LIN {X 0,Y 657.537,Z 599.865,A -85,B 0,C 180,E1 28395.268,E2 28395.268} C_VEL
LIN {X 0,Y 653.321,Z 821.185,A -85,B 0,C 180,E1 28392.316,E2 28392.316} C_VEL
LIN {X 0,Y 652.432,Z 844.585,A -85,B 0,C 180,E1 28391.93,E2 28391.93} C_VEL
LIN {X 0,Y 651.296,Z 867.25,A -85,B 0,C 180,E1 28391.436,E2 28391.436} C_VEL
LIN {X 0,Y 649.719,Z 893.344,A -85,B 0,C 180,E1 28390.715,E2 28390.715} C_VEL
LIN {X 0,Y 647.795,Z 918.743,A -85,B 0,C 180,E1 28389.832,E2 28389.832} C_VEL
LIN {X 0,Y 645.973,Z 940.605,A -85,B 0,C 180,E1 28388.933,E2 28388.933} C_VEL
LIN {X 0,Y 644.086,Z 961.718,A -85,B 0,C 180,E1 28387.933,E2 28387.933} C_VEL
LIN {X 0,Y 641.744,Z 986.523,A -85,B 0,C 180,E1 28386.58,E2 28386.58} C_VEL
LIN {X 0,Y 639.474,Z 1008.599,A -85,B 0,C 180,E1 28385.182,E2 28385.182} C_VEL
LIN {X 0,Y 637.565,Z 1026.909,A -85,B 0,C 180,E1 28383.884,E2 28383.884} C_VEL
LIN {X 0,Y 635.698,Z 1044.667,A -85,B 0,C 180,E1 28382.488,E2 28382.488} C_VEL
LIN {X 0,Y 633.545,Z 1065.498,A -85,B 0,C 180,E1 28380.667,E2 28380.667} C_VEL
LIN {X 0,Y 631.511,Z 1085.195,A -85,B 0,C 180,E1 28378.697,E2 28378.697} C_VEL
LIN {X 0,Y 630.035,Z 1100.537,A -85,B 0,C 180,E1 28376.993,E2 28376.993} C_VEL
LIN {X 0,Y 628.438,Z 1118.013,A -85,B 0,C 180,E1 28374.836,E2 28374.836} C_VEL
LIN {X 0,Y 627.118,Z 1133.831,A -85,B 0,C 180,E1 28372.597,E2 28372.597} C_VEL
LIN {X 0,Y 626.191,Z 1146.584,A -85,B 0,C 180,E1 28370.566,E2 28370.566} C_VEL
LIN {X 0,Y 625.357,Z 1159.892,A -85,B 0,C 180,E1 28368.166,E2 28368.166} C_VEL
LIN {X 0,Y 624.743,Z 1171.081,A -85,B 0,C 180,E1 28365.788,E2 28365.788} C_VEL
LIN {X 0,Y 624.416,Z 1179.161,A -85,B 0,C 180,E1 28363.803,E2 28363.803} C_VEL
LIN {X 0,Y 624.174,Z 1186.707,A -85,B 0,C 180,E1 28361.644,E2 28361.644} C_VEL
LIN {X 0,Y 624.016,Z 1193.595,A -85,B 0,C 180,E1 28359.22,E2 28359.22} C_VEL
LIN {X 0,Y 623.938,Z 1198.919,A -85,B 0,C 180,E1 28356.718,E2 28356.718} C_VEL
LIN {X 0,Y 623.914,Z 1202.24,A -85,B 0,C 180,E1 28354.504,E2 28354.504} C_VEL
LIN {X 0,Y 623.912,Z 1204.382,A -85,B 0,C 180,E1 28352.112,E2 28352.112} C_VEL
LIN {X 0,Y 623.892,Z 1204.894,A -85,B 0,C 180,E1 28349.541,E2 28349.541} C_VEL
LIN {X 0,Y 623.91,Z 1204.004,A -85,B 0,C 180,E1 28347.336,E2 28347.336} C_VEL
LIN {X 0,Y 623.923,Z 1201.671,A -85,B 0,C 180,E1 28345.036,E2 28345.036} C_VEL
LIN {X 0,Y 623.958,Z 1197.542,A -85,B 0,C 180,E1 28342.542,E2 28342.542} C_VEL
LIN {X 0,Y 624.046,Z 1191.872,A -85,B 0,C 180,E1 28340.129,E2 28340.129} C_VEL
LIN {X 0,Y 624.21,Z 1184.888,A -85,B 0,C 180,E1 28337.793,E2 28337.793} C_VEL
LIN {X 0,Y 624.578,Z 1175.442,A -85,B 0,C 180,E1 28335.229,E2 28335.229} C_VEL
LIN {X 0,Y 625.049,Z 1164.999,A -85,B 0,C 180,E1 28332.882,E2 28332.882} C_VEL
LIN {X 0,Y 625.664,Z 1154.466,A -85,B 0,C 180,E1 28330.821,E2 28330.821} C_VEL
LIN {X 0,Y 626.613,Z 1140.788,A -85,B 0,C 180,E1 28328.469,E2 28328.469} C_VEL
LIN {X 0,Y 627.822,Z 1125.096,A -85,B 0,C 180,E1 28326.139,E2 28326.139} C_VEL
LIN {X 0,Y 629.061,Z 1111.084,A -85,B 0,C 180,E1 28324.284,E2 28324.284} C_VEL
LIN {X 0,Y 630.771,Z 1092.863,A -85,B 0,C 180,E1 28322.12,E2 28322.12} C_VEL
LIN {X 0,Y 632.663,Z 1073.815,A -85,B 0,C 180,E1 28320.144,E2 28320.144} C_VEL
LIN {X 0,Y 634.36,Z 1057.393,A -85,B 0,C 180,E1 28318.606,E2 28318.606} C_VEL
LIN {X 0,Y 636.318,Z 1038.641,A -85,B 0,C 180,E1 28317.018,E2 28317.018} C_VEL
LIN {X 0,Y 638.857,Z 1014.539,A -85,B 0,C 180,E1 28315.223,E2 28315.223} C_VEL
LIN {X 0,Y 640.898,Z 994.594,A -85,B 0,C 180,E1 28313.916,E2 28313.916} C_VEL
LIN {X 0,Y 642.854,Z 974.951,A -85,B 0,C 180,E1 28312.769,E2 28312.769} C_VEL
LIN {X 0,Y 645.083,Z 951.673,A -85,B 0,C 180,E1 28311.572,E2 28311.572} C_VEL
LIN {X 0,Y 647.292,Z 925.381,A -85,B 0,C 180,E1 28310.428,E2 28310.428} C_VEL
LIN {X 0,Y 648.897,Z 904.132,A -85,B 0,C 180,E1 28309.643,E2 28309.643} C_VEL
LIN {X 0,Y 650.369,Z 882.585,A -85,B 0,C 180,E1 28308.97,E2 28308.97} C_VEL
LIN {X 0,Y 651.781,Z 858.661,A -85,B 0,C 180,E1 28308.36,E2 28308.36} C_VEL
LIN {X 0,Y 653.042,Z 830.092,A -85,B 0,C 180,E1 28307.816,E2 28307.816} C_VEL
LIN {X 0,Y 654.465,Z 762.422,A -85,B 0,C 180,E1 28306.902,E2 28306.902} C_VEL
LIN {X 0,Y 658.724,Z 539.813,A -85,B 0,C 180,E1 28303.919,E2 28303.919} C_VEL
LIN {X 0,Y 661.621,Z 393.143,A -85,B 0,C 180,E1 28301.897,E2 28301.897} C_VEL
LIN {X 0,Y 647.792,Z 372.953,A -85,B 0,C 180,E1 28300.181,E2 28300.181} C_VEL
LIN {X 0,Y 638.276,Z 359.45,A -85,B 0,C 180,E1 28298.917,E2 28298.917} C_VEL
LIN {X 0,Y 631.39,Z 349.683,A -85,B 0,C 180,E1 28297.912,E2 28297.912} C_VEL
LIN {X 0,Y 627.324,Z 341.452,A -85,B 0,C 180,E1 28296.593,E2 28296.593} C_VEL
LIN {X 0,Y 625.216,Z 337.776,A -85,B 0,C 180,E1 28295.94,E2 28295.94} C_VEL
LIN {X 0,Y 624.896,Z 336.388,A -85,B 0,C 180,E1 28295.735,E2 28295.735} C_VEL
LIN {X 0,Y 624.89,Z 336.391,A -85,B 0,C 180,E1 28292.959,E2 28292.959} C_VEL
LIN {X 0,Y 624.914,Z 336.381,A -85,B 0,C 180,E1 28289.737,E2 28289.737} C_VEL
LIN {X 0,Y 624.88,Z 336.358,A -85,B 0,C 180,E1 28286.97,E2 28286.97} C_VEL
LIN {X 0,Y 624.953,Z 336.372,A -85,B 0,C 180,E1 28283.878,E2 28283.878} C_VEL
LIN {X 0,Y 624.884,Z 336.384,A -85,B 0,C 180,E1 28280.906,E2 28280.906} C_VEL
LIN {X 0,Y 624.944,Z 336.356,A -85,B 0,C 180,E1 28277.987,E2 28277.987} C_VEL
LIN {X 0,Y 624.888,Z 336.391,A -85,B 0,C 180,E1 28274.887,E2 28274.887} C_VEL
LIN {X 0,Y 624.922,Z 336.352,A -85,B 0,C 180,E1 28272.005,E2 28272.005} C_VEL
LIN {X 0,Y 624.895,Z 336.385,A -85,B 0,C 180,E1 28268.836,E2 28268.836} C_VEL
LIN {X 0,Y 624.901,Z 336.36,A -85,B 0,C 180,E1 28266.062,E2 28266.062} C_VEL
LIN {X 0,Y 624.901,Z 336.375,A -85,B 0,C 180,E1 28262.751,E2 28262.751} C_VEL
LIN {X 0,Y 624.902,Z 336.375,A -85,B 0,C 180,E1 28259.908,E2 28259.908} C_VEL
LIN {X 0,Y 624.903,Z 336.36,A -85,B 0,C 180,E1 28256.606,E2 28256.606} C_VEL
LIN {X 0,Y 624.903,Z 336.384,A -85,B 0,C 180,E1 28253.754,E2 28253.754} C_VEL
LIN {X 0,Y 624.912,Z 336.355,A -85,B 0,C 180,E1 28250.514,E2 28250.514} C_VEL
LIN {X 0,Y 624.902,Z 336.388,A -85,B 0,C 180,E1 28247.619,E2 28247.619} C_VEL
LIN {X 0,Y 624.921,Z 336.363,A -85,B 0,C 180,E1 28244.404,E2 28244.404} C_VEL
LIN {X 0,Y 624.897,Z 336.37,A -85,B 0,C 180,E1 28241.529,E2 28241.529} C_VEL
LIN {X 0,Y 624.942,Z 336.389,A -85,B 0,C 180,E1 28238.365,E2 28238.365} C_VEL
LIN {X 0,Y 624.894,Z 336.369,A -85,B 0,C 180,E1 28235.416,E2 28235.416} C_VEL
LIN {X 0,Y 624.956,Z 336.386,A -85,B 0,C 180,E1 28232.355,E2 28232.355} C_VEL
LIN {X 0,Y 624.976,Z 336.514,A -85,B 0,C 180,E1 28230.372,E2 28230.372} C_VEL
LIN {X 0,Y 626.376,Z 340.092,A -85,B 0,C 180,E1 28229.812,E2 28229.812} C_VEL
LIN {X 0,Y 627.464,Z 341.921,A -85,B 0,C 180,E1 28229.499,E2 28229.499} C_VEL
LIN {X 0,Y 630.591,Z 346.07,A -85,B 0,C 180,E1 28229.033,E2 28229.033} C_VEL
LIN {X 0,Y 642.353,Z 362.019,A -85,B 0,C 180,E1 28227.386,E2 28227.386} C_VEL
LIN {X 0,Y 655.331,Z 380.655,A -85,B 0,C 180,E1 28225.722,E2 28225.722} C_VEL
LIN {X 0,Y 661.575,Z 390.24,A -85,B 0,C 180,E1 28224.954,E2 28224.954} C_VEL
LIN {X 0,Y 659.29,Z 501.464,A -85,B 0,C 180,E1 28223.422,E2 28223.422} C_VEL
LIN {X 0,Y 658.447,Z 509.169,A -85,B 0,C 180,E1 28223.38,E2 28223.38} C_VEL
LIN {X 0,Y 653.685,Z 529.837,A -85,B 0,C 180,E1 28223.497,E2 28223.497} C_VEL
LIN {X 0,Y 653.027,Z 536.446,A -85,B 0,C 180,E1 28223.454,E2 28223.454} C_VEL
LIN {X 0,Y 648.61,Z 753.058,A -85,B 0,C 180,E1 28220.529,E2 28220.529} C_VEL
LIN {X 0,Y 647.089,Z 821.836,A -85,B 0,C 180,E1 28219.592,E2 28219.592} C_VEL
LIN {X 0,Y 645.779,Z 848.344,A -85,B 0,C 180,E1 28219.075,E2 28219.075} C_VEL
LIN {X 0,Y 644.398,Z 870.837,A -85,B 0,C 180,E1 28218.507,E2 28218.507} C_VEL
LIN {X 0,Y 642.785,Z 893.737,A -85,B 0,C 180,E1 28217.797,E2 28217.797} C_VEL
LIN {X 0,Y 640.614,Z 920.334,A -85,B 0,C 180,E1 28216.793,E2 28216.793} C_VEL
LIN {X 0,Y 638.585,Z 942.122,A -85,B 0,C 180,E1 28215.816,E2 28215.816} C_VEL
LIN {X 0,Y 636.483,Z 963.279,A -85,B 0,C 180,E1 28214.73,E2 28214.73} C_VEL
LIN {X 0,Y 633.956,Z 987.267,A -85,B 0,C 180,E1 28213.32,E2 28213.32} C_VEL
LIN {X 0,Y 631.38,Z 1010.175,A -85,B 0,C 180,E1 28211.763,E2 28211.763} C_VEL
LIN {X 0,Y 628.962,Z 1032.056,A -85,B 0,C 180,E1 28210.078,E2 28210.078} C_VEL
LIN {X 0,Y 626.551,Z 1053.456,A -85,B 0,C 180,E1 28208.198,E2 28208.198} C_VEL
LIN {X 0,Y 624.312,Z 1073.834,A -85,B 0,C 180,E1 28206.176,E2 28206.176} C_VEL
LIN {X 0,Y 622.264,Z 1093.517,A -85,B 0,C 180,E1 28203.948,E2 28203.948} C_VEL
LIN {X 0,Y 620.561,Z 1111.006,A -85,B 0,C 180,E1 28201.706,E2 28201.706} C_VEL
LIN {X 0,Y 619.125,Z 1127.45,A -85,B 0,C 180,E1 28199.295,E2 28199.295} C_VEL
LIN {X 0,Y 618.008,Z 1142.104,A -85,B 0,C 180,E1 28196.833,E2 28196.833} C_VEL
LIN {X 0,Y 617.161,Z 1155.043,A -85,B 0,C 180,E1 28194.299,E2 28194.299} C_VEL
LIN {X 0,Y 616.625,Z 1165.506,A -85,B 0,C 180,E1 28191.897,E2 28191.897} C_VEL
LIN {X 0,Y 616.242,Z 1174.897,A -85,B 0,C 180,E1 28189.329,E2 28189.329} C_VEL
LIN {X 0,Y 616.066,Z 1181.779,A -85,B 0,C 180,E1 28186.986,E2 28186.986} C_VEL
LIN {X 0,Y 615.973,Z 1187.229,A -85,B 0,C 180,E1 28184.653,E2 28184.653} C_VEL
LIN {X 0,Y 615.925,Z 1191.546,A -85,B 0,C 180,E1 28182.088,E2 28182.088} C_VEL
LIN {X 0,Y 615.913,Z 1193.955,A -85,B 0,C 180,E1 28179.72,E2 28179.72} C_VEL
LIN {X 0,Y 615.896,Z 1194.864,A -85,B 0,C 180,E1 28177.556,E2 28177.556} C_VEL
LIN {X 0,Y 615.914,Z 1194.562,A -85,B 0,C 180,E1 28175.123,E2 28175.123} C_VEL
LIN {X 0,Y 615.916,Z 1192.49,A -85,B 0,C 180,E1 28172.605,E2 28172.605} C_VEL
LIN {X 0,Y 615.946,Z 1189.149,A -85,B 0,C 180,E1 28170.279,E2 28170.279} C_VEL
LIN {X 0,Y 616.031,Z 1183.731,A -85,B 0,C 180,E1 28167.675,E2 28167.675} C_VEL
LIN {X 0,Y 616.189,Z 1176.982,A -85,B 0,C 180,E1 28165.253,E2 28165.253} C_VEL
LIN {X 0,Y 616.445,Z 1169.355,A -85,B 0,C 180,E1 28163.013,E2 28163.013} C_VEL
LIN {X 0,Y 616.94,Z 1159.075,A -85,B 0,C 180,E1 28160.485,E2 28160.485} C_VEL
LIN {X 0,Y 617.683,Z 1146.755,A -85,B 0,C 180,E1 28157.947,E2 28157.947} C_VEL
LIN {X 0,Y 618.726,Z 1132.355,A -85,B 0,C 180,E1 28155.399,E2 28155.399} C_VEL
LIN {X 0,Y 620.085,Z 1116.227,A -85,B 0,C 180,E1 28152.934,E2 28152.934} C_VEL
LIN {X 0,Y 621.745,Z 1098.393,A -85,B 0,C 180,E1 28150.556,E2 28150.556} C_VEL
LIN {X 0,Y 623.702,Z 1079.651,A -85,B 0,C 180,E1 28148.364,E2 28148.364} C_VEL
LIN {X 0,Y 625.944,Z 1058.763,A -85,B 0,C 180,E1 28146.213,E2 28146.213} C_VEL
LIN {X 0,Y 628.328,Z 1037.643,A -85,B 0,C 180,E1 28144.302,E2 28144.302} C_VEL
LIN {X 0,Y 630.948,Z 1014.168,A -85,B 0,C 180,E1 28142.437,E2 28142.437} C_VEL
LIN {X 0,Y 633.461,Z 991.448,A -85,B 0,C 180,E1 28140.861,E2 28140.861} C_VEL
LIN {X 0,Y 636.2,Z 966.176,A -85,B 0,C 180,E1 28139.337,E2 28139.337} C_VEL
LIN {X 0,Y 638.384,Z 944.2,A -85,B 0,C 180,E1 28138.195,E2 28138.195} C_VEL
LIN {X 0,Y 640.435,Z 922.22,A -85,B 0,C 180,E1 28137.198,E2 28137.198} C_VEL
LIN {X 0,Y 642.615,Z 896.084,A -85,B 0,C 180,E1 28136.191,E2 28136.191} C_VEL
LIN {X 0,Y 644.347,Z 871.789,A -85,B 0,C 180,E1 28135.431,E2 28135.431} C_VEL
LIN {X 0,Y 645.709,Z 849.449,A -85,B 0,C 180,E1 28134.86,E2 28134.86} C_VEL
LIN {X 0,Y 646.986,Z 824.075,A -85,B 0,C 180,E1 28134.355,E2 28134.355} C_VEL
LIN {X 0,Y 648.108,Z 779.029,A -85,B 0,C 180,E1 28133.727,E2 28133.727} C_VEL
LIN {X 0,Y 652.675,Z 553.676,A -85,B 0,C 180,E1 28130.693,E2 28130.693} C_VEL
LIN {X 0,Y 656.073,Z 393.886,A -85,B 0,C 180,E1 28128.478,E2 28128.478} C_VEL
LIN {X 0,Y 644.814,Z 377.11,A -85,B 0,C 180,E1 28127.047,E2 28127.047} C_VEL
LIN {X 0,Y 633.812,Z 361.802,A -85,B 0,C 180,E1 28125.582,E2 28125.582} C_VEL
LIN {X 0,Y 626.174,Z 351.738,A -85,B 0,C 180,E1 28124.54,E2 28124.54} C_VEL
LIN {X 0,Y 622.262,Z 346.503,A -85,B 0,C 180,E1 28123.993,E2 28123.993} C_VEL
LIN {X 0,Y 618.866,Z 341.624,A -85,B 0,C 180,E1 28123.494,E2 28123.494} C_VEL
LIN {X 0,Y 617.209,Z 338.714,A -85,B 0,C 180,E1 28123.003,E2 28123.003} C_VEL
LIN {X 0,Y 616.913,Z 337.36,A -85,B 0,C 180,E1 28122.807,E2 28122.807} C_VEL
LIN {X 0,Y 616.952,Z 337.385,A -85,B 0,C 180,E1 28120.047,E2 28120.047} C_VEL
LIN {X 0,Y 616.924,Z 337.379,A -85,B 0,C 180,E1 28116.848,E2 28116.848} C_VEL
LIN {X 0,Y 616.932,Z 337.375,A -85,B 0,C 180,E1 28114.089,E2 28114.089} C_VEL
LIN {X 0,Y 616.933,Z 337.382,A -85,B 0,C 180,E1 28110.8,E2 28110.8} C_VEL
LIN {X 0,Y 616.92,Z 337.342,A -85,B 0,C 180,E1 28108.141,E2 28108.141} C_VEL
LIN {X 0,Y 616.979,Z 337.38,A -85,B 0,C 180,E1 28105.023,E2 28105.023} C_VEL
LIN {X 0,Y 616.916,Z 337.342,A -85,B 0,C 180,E1 28102.188,E2 28102.188} C_VEL
LIN {X 0,Y 616.993,Z 337.368,A -85,B 0,C 180,E1 28099.207,E2 28099.207} C_VEL
LIN {X 0,Y 616.923,Z 337.376,A -85,B 0,C 180,E1 28096.187,E2 28096.187} C_VEL
LIN {X 0,Y 616.941,Z 337.373,A -85,B 0,C 180,E1 28093.493,E2 28093.493} C_VEL
LIN {X 0,Y 616.939,Z 337.369,A -85,B 0,C 180,E1 28090.27,E2 28090.27} C_VEL
LIN {X 0,Y 616.931,Z 337.381,A -85,B 0,C 180,E1 28087.544,E2 28087.544} C_VEL
LIN {X 0,Y 616.981,Z 337.377,A -85,B 0,C 180,E1 28084.462,E2 28084.462} C_VEL
LIN {X 0,Y 616.924,Z 337.377,A -85,B 0,C 180,E1 28081.579,E2 28081.579} C_VEL
LIN {X 0,Y 617.008,Z 337.365,A -85,B 0,C 180,E1 28078.607,E2 28078.607} C_VEL
LIN {X 0,Y 616.926,Z 337.368,A -85,B 0,C 180,E1 28075.538,E2 28075.538} C_VEL
LIN {X 0,Y 616.981,Z 337.371,A -85,B 0,C 180,E1 28072.644,E2 28072.644} C_VEL
LIN {X 0,Y 616.934,Z 337.376,A -85,B 0,C 180,E1 28069.541,E2 28069.541} C_VEL
LIN {X 0,Y 616.953,Z 337.333,A -85,B 0,C 180,E1 28066.695,E2 28066.695} C_VEL
LIN {X 0,Y 616.945,Z 337.378,A -85,B 0,C 180,E1 28063.523,E2 28063.523} C_VEL
LIN {X 0,Y 616.934,Z 337.337,A -85,B 0,C 180,E1 28060.791,E2 28060.791} C_VEL
LIN {X 0,Y 616.97,Z 337.375,A -85,B 0,C 180,E1 28057.613,E2 28057.613} C_VEL
LIN {X 0,Y 616.931,Z 337.34,A -85,B 0,C 180,E1 28054.77,E2 28054.77} C_VEL
LIN {X 0,Y 616.996,Z 337.367,A -85,B 0,C 180,E1 28051.635,E2 28051.635} C_VEL
LIN {X 0,Y 616.934,Z 337.374,A -85,B 0,C 180,E1 28048.759,E2 28048.759} C_VEL
LIN {X 0,Y 617.011,Z 337.376,A -85,B 0,C 180,E1 28045.735,E2 28045.735} C_VEL
LIN {X 0,Y 616.961,Z 337.53,A -85,B 0,C 180,E1 28044.876,E2 28044.876} C_VEL
LIN {X 0,Y 618.247,Z 340.864,A -85,B 0,C 180,E1 28044.392,E2 28044.392} C_VEL
LIN {X 0,Y 619.292,Z 342.381,A -85,B 0,C 180,E1 28044.12,E2 28044.12} C_VEL
LIN {X 0,Y 623.249,Z 350.426,A -85,B 0,C 180,E1 28042.927,E2 28042.927} C_VEL
LIN {X 0,Y 633.099,Z 363.839,A -85,B 0,C 180,E1 28041.57,E2 28041.57} C_VEL
LIN {X 0,Y 642.371,Z 376.815,A -85,B 0,C 180,E1 28040.328,E2 28040.328} C_VEL
LIN {X 0,Y 654.585,Z 394.719,A -85,B 0,C 180,E1 28038.767,E2 28038.767} C_VEL
LIN {X 0,Y 656.243,Z 397.52,A -85,B 0,C 180,E1 28038.557,E2 28038.557} C_VEL
LIN {X 0,Y 651.839,Z 602.931,A -85,B 0,C 180,E1 28035.728,E2 28035.728} C_VEL
LIN {X 0,Y 647.36,Z 822.437,A -85,B 0,C 180,E1 28032.775,E2 28032.775} C_VEL
LIN {X 0,Y 646.442,Z 845.047,A -85,B 0,C 180,E1 28032.397,E2 28032.397} C_VEL
LIN {X 0,Y 645.242,Z 867.553,A -85,B 0,C 180,E1 28031.903,E2 28031.903} C_VEL
LIN {X 0,Y 643.563,Z 893.754,A -85,B 0,C 180,E1 28031.174,E2 28031.174} C_VEL
LIN {X 0,Y 641.555,Z 918.74,A -85,B 0,C 180,E1 28030.299,E2 28030.299} C_VEL
LIN {X 0,Y 639.694,Z 939.866,A -85,B 0,C 180,E1 28029.427,E2 28029.427} C_VEL
LIN {X 0,Y 637.715,Z 960.71,A -85,B 0,C 180,E1 28028.437,E2 28028.437} C_VEL
LIN {X 0,Y 635.358,Z 983.923,A -85,B 0,C 180,E1 28027.178,E2 28027.178} C_VEL
LIN {X 0,Y 632.763,Z 1007.862,A -85,B 0,C 180,E1 28025.667,E2 28025.667} C_VEL
LIN {X 0,Y 630.635,Z 1026.957,A -85,B 0,C 180,E1 28024.303,E2 28024.303} C_VEL
LIN {X 0,Y 628.619,Z 1044.936,A -85,B 0,C 180,E1 28022.876,E2 28022.876} C_VEL
LIN {X 0,Y 626.328,Z 1065.691,A -85,B 0,C 180,E1 28021.04,E2 28021.04} C_VEL
LIN {X 0,Y 624.159,Z 1084.994,A -85,B 0,C 180,E1 28019.09,E2 28019.09} C_VEL
LIN {X 0,Y 622.55,Z 1100.535,A -85,B 0,C 180,E1 28017.344,E2 28017.344} C_VEL
LIN {X 0,Y 620.832,Z 1118.042,A -85,B 0,C 180,E1 28015.158,E2 28015.158} C_VEL
LIN {X 0,Y 619.41,Z 1133.833,A -85,B 0,C 180,E1 28012.894,E2 28012.894} C_VEL
LIN {X 0,Y 618.402,Z 1146.582,A -85,B 0,C 180,E1 28010.837,E2 28010.837} C_VEL
LIN {X 0,Y 617.488,Z 1159.949,A -85,B 0,C 180,E1 28008.394,E2 28008.394} C_VEL
LIN {X 0,Y 616.833,Z 1171.082,A -85,B 0,C 180,E1 28005.995,E2 28005.995} C_VEL
LIN {X 0,Y 616.461,Z 1179.162,A -85,B 0,C 180,E1 28003.985,E2 28003.985} C_VEL
LIN {X 0,Y 616.199,Z 1186.401,A -85,B 0,C 180,E1 28001.892,E2 28001.892} C_VEL
LIN {X 0,Y 616.035,Z 1193.353,A -85,B 0,C 180,E1 27999.435,E2 27999.435} C_VEL
LIN {X 0,Y 615.943,Z 1198.756,A -85,B 0,C 180,E1 27996.899,E2 27996.899} C_VEL
LIN {X 0,Y 615.914,Z 1202.2,A -85,B 0,C 180,E1 27994.593,E2 27994.593} C_VEL
LIN {X 0,Y 615.911,Z 1204.326,A -85,B 0,C 180,E1 27992.233,E2 27992.233} C_VEL
LIN {X 0,Y 615.894,Z 1204.917,A -85,B 0,C 180,E1 27989.628,E2 27989.628} C_VEL
LIN {X 0,Y 615.911,Z 1204.001,A -85,B 0,C 180,E1 27987.302,E2 27987.302} C_VEL
LIN {X 0,Y 615.925,Z 1201.668,A -85,B 0,C 180,E1 27984.971,E2 27984.971} C_VEL
LIN {X 0,Y 615.96,Z 1197.542,A -85,B 0,C 180,E1 27982.445,E2 27982.445} C_VEL
LIN {X 0,Y 616.061,Z 1191.869,A -85,B 0,C 180,E1 27979.999,E2 27979.999} C_VEL
LIN {X 0,Y 616.231,Z 1185.188,A -85,B 0,C 180,E1 27977.728,E2 27977.728} C_VEL
LIN {X 0,Y 616.603,Z 1176.301,A -85,B 0,C 180,E1 27975.251,E2 27975.251} C_VEL
LIN {X 0,Y 617.134,Z 1165.456,A -85,B 0,C 180,E1 27972.753,E2 27972.753} C_VEL
LIN {X 0,Y 617.794,Z 1154.968,A -85,B 0,C 180,E1 27970.662,E2 27970.662} C_VEL
LIN {X 0,Y 618.708,Z 1142.537,A -85,B 0,C 180,E1 27968.479,E2 27968.479} C_VEL
LIN {X 0,Y 620.047,Z 1126.495,A -85,B 0,C 180,E1 27966.023,E2 27966.023} C_VEL
LIN {X 0,Y 621.426,Z 1111.852,A -85,B 0,C 180,E1 27964.047,E2 27964.047} C_VEL
LIN {X 0,Y 623.059,Z 1095.44,A -85,B 0,C 180,E1 27962.057,E2 27962.057} C_VEL
LIN {X 0,Y 625.236,Z 1075.26,A -85,B 0,C 180,E1 27959.904,E2 27959.904} C_VEL
LIN {X 0,Y 627.085,Z 1058.502,A -85,B 0,C 180,E1 27958.307,E2 27958.307} C_VEL
LIN {X 0,Y 629.038,Z 1041.012,A -85,B 0,C 180,E1 27956.799,E2 27956.799} C_VEL
LIN {X 0,Y 631.555,Z 1018.937,A -85,B 0,C 180,E1 27955.096,E2 27955.096} C_VEL
LIN {X 0,Y 634.035,Z 996.25,A -85,B 0,C 180,E1 27953.578,E2 27953.578} C_VEL
LIN {X 0,Y 636.01,Z 977.648,A -85,B 0,C 180,E1 27952.47,E2 27952.47} C_VEL
LIN {X 0,Y 638.028,Z 957.699,A -85,B 0,C 180,E1 27951.413,E2 27951.413} C_VEL
LIN {X 0,Y 640.077,Z 936.082,A -85,B 0,C 180,E1 27950.407,E2 27950.407} C_VEL
LIN {X 0,Y 642.391,Z 908.567,A -85,B 0,C 180,E1 27949.325,E2 27949.325} C_VEL
LIN {X 0,Y 644.095,Z 885.248,A -85,B 0,C 180,E1 27948.574,E2 27948.574} C_VEL
LIN {X 0,Y 645.474,Z 863.386,A -85,B 0,C 180,E1 27947.996,E2 27947.996} C_VEL
LIN {X 0,Y 646.71,Z 839.526,A -85,B 0,C 180,E1 27947.497,E2 27947.497} C_VEL
LIN {X 0,Y 647.823,Z 804.077,A -85,B 0,C 180,E1 27946.972,E2 27946.972} C_VEL
LIN {X 0,Y 652.338,Z 579.129,A -85,B 0,C 180,E1 27943.949,E2 27943.949} C_VEL
LIN {X 0,Y 656.196,Z 397.117,A -85,B 0,C 180,E1 27941.433,E2 27941.433} C_VEL
LIN {X 0,Y 643.844,Z 378.961,A -85,B 0,C 180,E1 27939.867,E2 27939.867} C_VEL
LIN {X 0,Y 634.511,Z 365.563,A -85,B 0,C 180,E1 27938.594,E2 27938.594} C_VEL
LIN {X 0,Y 627.301,Z 355.568,A -85,B 0,C 180,E1 27937.538,E2 27937.538} C_VEL
LIN {X 0,Y 622.667,Z 349.349,A -85,B 0,C 180,E1 27936.796,E2 27936.796} C_VEL
LIN {X 0,Y 621.071,Z 345.95,A -85,B 0,C 180,E1 27936.239,E2 27936.239} C_VEL
LIN {X 0,Y 619.099,Z 341.914,A -85,B 0,C 180,E1 27935.551,E2 27935.551} C_VEL
LIN {X 0,Y 617.239,Z 338.715,A -85,B 0,C 180,E1 27934.949,E2 27934.949} C_VEL
LIN {X 0,Y 616.972,Z 337.377,A -85,B 0,C 180,E1 27934.751,E2 27934.751} C_VEL
LIN {X 0,Y 616.947,Z 337.347,A -85,B 0,C 180,E1 27931.52,E2 27931.52} C_VEL
LIN {X 0,Y 616.958,Z 337.378,A -85,B 0,C 180,E1 27928.747,E2 27928.747} C_VEL
LIN {X 0,Y 616.961,Z 337.371,A -85,B 0,C 180,E1 27925.435,E2 27925.435} C_VEL
LIN {X 0,Y 616.949,Z 337.346,A -85,B 0,C 180,E1 27922.689,E2 27922.689} C_VEL
LIN {X 0,Y 616.986,Z 337.373,A -85,B 0,C 180,E1 27919.502,E2 27919.502} C_VEL
LIN {X 0,Y 616.948,Z 337.354,A -85,B 0,C 180,E1 27916.574,E2 27916.574} C_VEL
LIN {X 0,Y 617.005,Z 337.353,A -85,B 0,C 180,E1 27913.495,E2 27913.495} C_VEL
LIN {X 0,Y 616.946,Z 337.373,A -85,B 0,C 180,E1 27910.553,E2 27910.553} C_VEL
LIN {X 0,Y 617.017,Z 337.342,A -85,B 0,C 180,E1 27907.543,E2 27907.543} C_VEL
LIN {X 0,Y 616.948,Z 337.379,A -85,B 0,C 180,E1 27904.462,E2 27904.462} C_VEL
LIN {X 0,Y 617.014,Z 337.337,A -85,B 0,C 180,E1 27901.393,E2 27901.393} C_VEL
LIN {X 0,Y 616.951,Z 337.378,A -85,B 0,C 180,E1 27898.328,E2 27898.328} C_VEL
LIN {X 0,Y 617.009,Z 337.336,A -85,B 0,C 180,E1 27895.259,E2 27895.259} C_VEL
LIN {X 0,Y 616.952,Z 337.371,A -85,B 0,C 180,E1 27892.175,E2 27892.175} C_VEL
LIN {X 0,Y 617.01,Z 337.354,A -85,B 0,C 180,E1 27889.117,E2 27889.117} C_VEL
LIN {X 0,Y 616.95,Z 337.349,A -85,B 0,C 180,E1 27886.026,E2 27886.026} C_VEL
LIN {X 0,Y 617.007,Z 337.373,A -85,B 0,C 180,E1 27883.04,E2 27883.04} C_VEL
LIN {X 0,Y 616.957,Z 337.353,A -85,B 0,C 180,E1 27879.904,E2 27879.904} C_VEL
LIN {X 0,Y 616.993,Z 337.351,A -85,B 0,C 180,E1 27876.993,E2 27876.993} C_VEL
LIN {X 0,Y 616.968,Z 337.375,A -85,B 0,C 180,E1 27873.844,E2 27873.844} C_VEL
LIN {X 0,Y 616.977,Z 337.512,A -85,B 0,C 180,E1 27871.36,E2 27871.36} C_VEL
LIN {X 0,Y 618.428,Z 341.031,A -85,B 0,C 180,E1 27870.772,E2 27870.772} C_VEL
LIN {X 0,Y 619.695,Z 342.64,A -85,B 0,C 180,E1 27870.493,E2 27870.493} C_VEL
LIN {X 0,Y 622.698,Z 346.846,A -85,B 0,C 180,E1 27870.014,E2 27870.014} C_VEL
LIN {X 0,Y 624.368,Z 348.918,A -85,B 0,C 180,E1 27869.758,E2 27869.758} C_VEL
LIN {X 0,Y 631.806,Z 358.777,A -85,B 0,C 180,E1 27868.649,E2 27868.649} C_VEL
LIN {X 0,Y 641.998,Z 373.086,A -85,B 0,C 180,E1 27867.233,E2 27867.233} C_VEL
LIN {X 0,Y 653.41,Z 389.714,A -85,B 0,C 180,E1 27865.767,E2 27865.767} C_VEL
LIN {X 0,Y 656.139,Z 394.138,A -85,B 0,C 180,E1 27865.422,E2 27865.422} C_VEL
LIN {X 0,Y 653.027,Z 536.446,A -85,B 0,C 180,E1 27863.454,E2 27863.454} C_VEL
LIN {X 0,Y 652.172,Z 544.153,A -85,B 0,C 180,E1 27863.412,E2 27863.412} C_VEL
LIN {X 0,Y 647.391,Z 564.821,A -85,B 0,C 180,E1 27863.532,E2 27863.532} C_VEL
LIN {X 0,Y 646.744,Z 571.43,A -85,B 0,C 180,E1 27863.488,E2 27863.488} C_VEL
LIN {X 0,Y 641.955,Z 794.936,A -85,B 0,C 180,E1 27860.461,E2 27860.461} C_VEL
LIN {X 0,Y 640.842,Z 828.606,A -85,B 0,C 180,E1 27859.959,E2 27859.959} C_VEL
LIN {X 0,Y 639.639,Z 851.198,A -85,B 0,C 180,E1 27859.493,E2 27859.493} C_VEL
LIN {X 0,Y 638.184,Z 873.466,A -85,B 0,C 180,E1 27858.914,E2 27858.914} C_VEL
LIN {X 0,Y 636.164,Z 899.915,A -85,B 0,C 180,E1 27858.063,E2 27858.063} C_VEL
LIN {X 0,Y 633.975,Z 924.132,A -85,B 0,C 180,E1 27857.102,E2 27857.102} C_VEL
LIN {X 0,Y 631.977,Z 944.368,A -85,B 0,C 180,E1 27856.174,E2 27856.174} C_VEL
LIN {X 0,Y 629.564,Z 967.293,A -85,B 0,C 180,E1 27854.97,E2 27854.97} C_VEL
LIN {X 0,Y 626.672,Z 992.212,A -85,B 0,C 180,E1 27853.445,E2 27853.445} C_VEL
LIN {X 0,Y 624.102,Z 1014.017,A -85,B 0,C 180,E1 27851.918,E2 27851.918} C_VEL
LIN {X 0,Y 621.349,Z 1037.166,A -85,B 0,C 180,E1 27850.066,E2 27850.066} C_VEL
LIN {X 0,Y 618.913,Z 1057.392,A -85,B 0,C 180,E1 27848.224,E2 27848.224} C_VEL
LIN {X 0,Y 616.558,Z 1077.724,A -85,B 0,C 180,E1 27846.135,E2 27846.135} C_VEL
LIN {X 0,Y 614.449,Z 1096.558,A -85,B 0,C 180,E1 27843.927,E2 27843.927} C_VEL
LIN {X 0,Y 612.722,Z 1113.396,A -85,B 0,C 180,E1 27841.698,E2 27841.698} C_VEL
LIN {X 0,Y 611.286,Z 1128.725,A -85,B 0,C 180,E1 27839.386,E2 27839.386} C_VEL
LIN {X 0,Y 610.149,Z 1142.652,A -85,B 0,C 180,E1 27836.996,E2 27836.996} C_VEL
LIN {X 0,Y 609.285,Z 1155.041,A -85,B 0,C 180,E1 27834.531,E2 27834.531} C_VEL
LIN {X 0,Y 608.694,Z 1165.506,A -85,B 0,C 180,E1 27832.096,E2 27832.096} C_VEL
LIN {X 0,Y 608.276,Z 1174.899,A -85,B 0,C 180,E1 27829.492,E2 27829.492} C_VEL
LIN {X 0,Y 608.077,Z 1181.781,A -85,B 0,C 180,E1 27827.117,E2 27827.117} C_VEL
LIN {X 0,Y 607.978,Z 1187.236,A -85,B 0,C 180,E1 27824.751,E2 27824.751} C_VEL
LIN {X 0,Y 607.927,Z 1191.549,A -85,B 0,C 180,E1 27822.153,E2 27822.153} C_VEL
LIN {X 0,Y 607.913,Z 1193.954,A -85,B 0,C 180,E1 27819.753,E2 27819.753} C_VEL
LIN {X 0,Y 607.896,Z 1194.864,A -85,B 0,C 180,E1 27817.561,E2 27817.561} C_VEL
LIN {X 0,Y 607.914,Z 1194.561,A -85,B 0,C 180,E1 27815.095,E2 27815.095} C_VEL
LIN {X 0,Y 607.916,Z 1192.594,A -85,B 0,C 180,E1 27812.64,E2 27812.64} C_VEL
LIN {X 0,Y 607.947,Z 1189.297,A -85,B 0,C 180,E1 27810.283,E2 27810.283} C_VEL
LIN {X 0,Y 608.033,Z 1184.177,A -85,B 0,C 180,E1 27807.738,E2 27807.738} C_VEL
LIN {X 0,Y 608.199,Z 1177.554,A -85,B 0,C 180,E1 27805.285,E2 27805.285} C_VEL
LIN {X 0,Y 608.47,Z 1170.001,A -85,B 0,C 180,E1 27803.002,E2 27803.002} C_VEL
LIN {X 0,Y 608.964,Z 1160.292,A -85,B 0,C 180,E1 27800.55,E2 27800.55} C_VEL
LIN {X 0,Y 609.696,Z 1148.69,A -85,B 0,C 180,E1 27798.075,E2 27798.075} C_VEL
LIN {X 0,Y 610.681,Z 1135.744,A -85,B 0,C 180,E1 27795.686,E2 27795.686} C_VEL
LIN {X 0,Y 611.983,Z 1120.791,A -85,B 0,C 180,E1 27793.289,E2 27793.289} C_VEL
LIN {X 0,Y 613.719,Z 1103.668,A -85,B 0,C 180,E1 27790.885,E2 27790.885} C_VEL
LIN {X 0,Y 615.645,Z 1085.617,A -85,B 0,C 180,E1 27788.667,E2 27788.667} C_VEL
LIN {X 0,Y 617.894,Z 1066.055,A -85,B 0,C 180,E1 27786.543,E2 27786.543} C_VEL
LIN {X 0,Y 620.44,Z 1044.529,A -85,B 0,C 180,E1 27784.488,E2 27784.488} C_VEL
LIN {X 0,Y 622.983,Z 1023.571,A -85,B 0,C 180,E1 27782.729,E2 27782.729} C_VEL
LIN {X 0,Y 625.786,Z 1000.122,A -85,B 0,C 180,E1 27780.993,E2 27780.993} C_VEL
LIN {X 0,Y 628.336,Z 977.646,A -85,B 0,C 180,E1 27779.548,E2 27779.548} C_VEL
LIN {X 0,Y 630.996,Z 953.824,A -85,B 0,C 180,E1 27778.206,E2 27778.206} C_VEL
LIN {X 0,Y 633.518,Z 928.818,A -85,B 0,C 180,E1 27777.01,E2 27777.01} C_VEL
LIN {X 0,Y 635.531,Z 906.678,A -85,B 0,C 180,E1 27776.102,E2 27776.102} C_VEL
LIN {X 0,Y 637.542,Z 882.584,A -85,B 0,C 180,E1 27775.268,E2 27775.268} C_VEL
LIN {X 0,Y 639.415,Z 854.875,A -85,B 0,C 180,E1 27774.502,E2 27774.502} C_VEL
LIN {X 0,Y 640.655,Z 832.174,A -85,B 0,C 180,E1 27774.017,E2 27774.017} C_VEL
LIN {X 0,Y 641.699,Z 806.596,A -85,B 0,C 180,E1 27773.606,E2 27773.606} C_VEL
LIN {X 0,Y 646.429,Z 585.413,A -85,B 0,C 180,E1 27770.614,E2 27770.614} C_VEL
LIN {X 0,Y 650.724,Z 397.897,A -85,B 0,C 180,E1 27768.008,E2 27768.008} C_VEL
LIN {X 0,Y 641.055,Z 383.358,A -85,B 0,C 180,E1 27766.753,E2 27766.753} C_VEL
LIN {X 0,Y 629.677,Z 367.481,A -85,B 0,C 180,E1 27765.22,E2 27765.22} C_VEL
LIN {X 0,Y 622.205,Z 357.667,A -85,B 0,C 180,E1 27764.19,E2 27764.19} C_VEL
LIN {X 0,Y 617.898,Z 351.945,A -85,B 0,C 180,E1 27763.58,E2 27763.58} C_VEL
LIN {X 0,Y 615.027,Z 347.904,A -85,B 0,C 180,E1 27763.161,E2 27763.161} C_VEL
LIN {X 0,Y 611.884,Z 343.756,A -85,B 0,C 180,E1 27762.7,E2 27762.7} C_VEL
LIN {X 0,Y 609.932,Z 341.243,A -85,B 0,C 180,E1 27762.359,E2 27762.359} C_VEL
LIN {X 0,Y 609.031,Z 338.336,A -85,B 0,C 180,E1 27761.929,E2 27761.929} C_VEL
LIN {X 0,Y 608.982,Z 338.37,A -85,B 0,C 180,E1 27758.845,E2 27758.845} C_VEL
LIN {X 0,Y 608.997,Z 338.371,A -85,B 0,C 180,E1 27756.117,E2 27756.117} C_VEL
LIN {X 0,Y 608.99,Z 338.369,A -85,B 0,C 180,E1 27752.808,E2 27752.808} C_VEL
LIN {X 0,Y 608.993,Z 338.371,A -85,B 0,C 180,E1 27750.051,E2 27750.051} C_VEL
LIN {X 0,Y 608.997,Z 338.339,A -85,B 0,C 180,E1 27746.729,E2 27746.729} C_VEL
LIN {X 0,Y 608.99,Z 338.369,A -85,B 0,C 180,E1 27743.925,E2 27743.925} C_VEL
LIN {X 0,Y 609.016,Z 338.329,A -85,B 0,C 180,E1 27740.771,E2 27740.771} C_VEL
LIN {X 0,Y 608.983,Z 338.37,A -85,B 0,C 180,E1 27737.98,E2 27737.98} C_VEL
LIN {X 0,Y 609.071,Z 338.365,A -85,B 0,C 180,E1 27734.936,E2 27734.936} C_VEL
LIN {X 0,Y 608.983,Z 338.369,A -85,B 0,C 180,E1 27731.892,E2 27731.892} C_VEL
LIN {X 0,Y 609.066,Z 338.358,A -85,B 0,C 180,E1 27728.79,E2 27728.79} C_VEL
LIN {X 0,Y 608.986,Z 338.36,A -85,B 0,C 180,E1 27725.843,E2 27725.843} C_VEL
LIN {X 0,Y 609.038,Z 338.357,A -85,B 0,C 180,E1 27722.917,E2 27722.917} C_VEL
LIN {X 0,Y 608.991,Z 338.364,A -85,B 0,C 180,E1 27719.812,E2 27719.812} C_VEL
LIN {X 0,Y 609.006,Z 338.37,A -85,B 0,C 180,E1 27717.083,E2 27717.083} C_VEL
LIN {X 0,Y 609.002,Z 338.369,A -85,B 0,C 180,E1 27713.779,E2 27713.779} C_VEL
LIN {X 0,Y 609,Z 338.365,A -85,B 0,C 180,E1 27711.027,E2 27711.027} C_VEL
LIN {X 0,Y 609.011,Z 338.325,A -85,B 0,C 180,E1 27707.772,E2 27707.772} C_VEL
LIN {X 0,Y 608.996,Z 338.361,A -85,B 0,C 180,E1 27704.965,E2 27704.965} C_VEL
LIN {X 0,Y 609.04,Z 338.33,A -85,B 0,C 180,E1 27701.824,E2 27701.824} C_VEL
LIN {X 0,Y 608.994,Z 338.363,A -85,B 0,C 180,E1 27698.926,E2 27698.926} C_VEL
LIN {X 0,Y 609.065,Z 338.321,A -85,B 0,C 180,E1 27695.872,E2 27695.872} C_VEL
LIN {X 0,Y 608.996,Z 338.37,A -85,B 0,C 180,E1 27692.842,E2 27692.842} C_VEL
LIN {X 0,Y 609.078,Z 338.36,A -85,B 0,C 180,E1 27689.845,E2 27689.845} C_VEL
LIN {X 0,Y 608.996,Z 338.362,A -85,B 0,C 180,E1 27686.744,E2 27686.744} C_VEL
LIN {X 0,Y 609.091,Z 338.512,A -85,B 0,C 180,E1 27685.76,E2 27685.76} C_VEL
LIN {X 0,Y 610.405,Z 341.953,A -85,B 0,C 180,E1 27685.246,E2 27685.246} C_VEL
LIN {X 0,Y 611.373,Z 343.545,A -85,B 0,C 180,E1 27684.966,E2 27684.966} C_VEL
LIN {X 0,Y 613.145,Z 347.109,A -85,B 0,C 180,E1 27684.396,E2 27684.396} C_VEL
LIN {X 0,Y 614.776,Z 350.335,A -85,B 0,C 180,E1 27683.93,E2 27683.93} C_VEL
LIN {X 0,Y 628.771,Z 369.174,A -85,B 0,C 180,E1 27681.96,E2 27681.96} C_VEL
LIN {X 0,Y 638.943,Z 383.551,A -85,B 0,C 180,E1 27680.582,E2 27680.582} C_VEL
LIN {X 0,Y 650.575,Z 400.712,A -85,B 0,C 180,E1 27679.071,E2 27679.071} C_VEL
LIN {X 0,Y 650.836,Z 401.888,A -85,B 0,C 180,E1 27679.025,E2 27679.025} C_VEL
LIN {X 0,Y 646.168,Z 606.309,A -85,B 0,C 180,E1 27676.191,E2 27676.191} C_VEL
LIN {X 0,Y 641.472,Z 822.833,A -85,B 0,C 180,E1 27673.256,E2 27673.256} C_VEL
LIN {X 0,Y 640.511,Z 845.184,A -85,B 0,C 180,E1 27672.88,E2 27672.88} C_VEL
LIN {X 0,Y 639.271,Z 867.168,A -85,B 0,C 180,E1 27672.395,E2 27672.395} C_VEL
LIN {X 0,Y 637.537,Z 892.934,A -85,B 0,C 180,E1 27671.679,E2 27671.679} C_VEL
LIN {X 0,Y 635.36,Z 918.737,A -85,B 0,C 180,E1 27670.774,E2 27670.774} C_VEL
LIN {X 0,Y 633.39,Z 939.906,A -85,B 0,C 180,E1 27669.895,E2 27669.895} C_VEL
LIN {X 0,Y 631.406,Z 959.702,A -85,B 0,C 180,E1 27668.952,E2 27668.952} C_VEL
LIN {X 0,Y 629.168,Z 980.481,A -85,B 0,C 180,E1 27667.829,E2 27667.829} C_VEL
LIN {X 0,Y 626.28,Z 1005.605,A -85,B 0,C 180,E1 27666.268,E2 27666.268} C_VEL
LIN {X 0,Y 623.824,Z 1026.236,A -85,B 0,C 180,E1 27664.791,E2 27664.791} C_VEL
LIN {X 0,Y 621.693,Z 1044.055,A -85,B 0,C 180,E1 27663.369,E2 27663.369} C_VEL
LIN {X 0,Y 619.498,Z 1062.618,A -85,B 0,C 180,E1 27661.723,E2 27661.723} C_VEL
LIN {X 0,Y 616.946,Z 1083.983,A -85,B 0,C 180,E1 27659.58,E2 27659.58} C_VEL
LIN {X 0,Y 615.165,Z 1099.687,A -85,B 0,C 180,E1 27657.806,E2 27657.806} C_VEL
LIN {X 0,Y 613.493,Z 1115.703,A -85,B 0,C 180,E1 27655.795,E2 27655.795} C_VEL
LIN {X 0,Y 611.778,Z 1133.19,A -85,B 0,C 180,E1 27653.298,E2 27653.298} C_VEL
LIN {X 0,Y 610.663,Z 1146.007,A -85,B 0,C 180,E1 27651.214,E2 27651.214} C_VEL
LIN {X 0,Y 609.727,Z 1158.363,A -85,B 0,C 180,E1 27648.947,E2 27648.947} C_VEL
LIN {X 0,Y 608.944,Z 1170.673,A -85,B 0,C 180,E1 27646.306,E2 27646.306} C_VEL
LIN {X 0,Y 608.513,Z 1179.162,A -85,B 0,C 180,E1 27644.171,E2 27644.171} C_VEL
LIN {X 0,Y 608.219,Z 1186.572,A -85,B 0,C 180,E1 27641.995,E2 27641.995} C_VEL
LIN {X 0,Y 608.042,Z 1193.595,A -85,B 0,C 180,E1 27639.465,E2 27639.465} C_VEL
LIN {X 0,Y 607.944,Z 1198.913,A -85,B 0,C 180,E1 27636.896,E2 27636.896} C_VEL
LIN {X 0,Y 607.914,Z 1202.234,A -85,B 0,C 180,E1 27634.623,E2 27634.623} C_VEL
LIN {X 0,Y 607.911,Z 1204.382,A -85,B 0,C 180,E1 27632.168,E2 27632.168} C_VEL
LIN {X 0,Y 607.893,Z 1204.894,A -85,B 0,C 180,E1 27629.529,E2 27629.529} C_VEL
LIN {X 0,Y 607.912,Z 1203.998,A -85,B 0,C 180,E1 27627.266,E2 27627.266} C_VEL
LIN {X 0,Y 607.924,Z 1201.779,A -85,B 0,C 180,E1 27624.999,E2 27624.999} C_VEL
LIN {X 0,Y 607.963,Z 1197.735,A -85,B 0,C 180,E1 27622.44,E2 27622.44} C_VEL
LIN {X 0,Y 608.07,Z 1192.121,A -85,B 0,C 180,E1 27619.962,E2 27619.962} C_VEL
LIN {X 0,Y 608.253,Z 1185.488,A -85,B 0,C 180,E1 27617.661,E2 27617.661} C_VEL
LIN {X 0,Y 608.607,Z 1177.374,A -85,B 0,C 180,E1 27615.345,E2 27615.345} C_VEL
LIN {X 0,Y 609.192,Z 1166.372,A -85,B 0,C 180,E1 27612.718,E2 27612.718} C_VEL
LIN {X 0,Y 609.902,Z 1155.793,A -85,B 0,C 180,E1 27610.562,E2 27610.562} C_VEL
LIN {X 0,Y 610.802,Z 1144.285,A -85,B 0,C 180,E1 27608.489,E2 27608.489} C_VEL
LIN {X 0,Y 612.149,Z 1129.295,A -85,B 0,C 180,E1 27606.104,E2 27606.104} C_VEL
LIN {X 0,Y 613.765,Z 1112.975,A -85,B 0,C 180,E1 27603.85,E2 27603.85} C_VEL
LIN {X 0,Y 615.429,Z 1097.312,A -85,B 0,C 180,E1 27601.911,E2 27601.911} C_VEL
LIN {X 0,Y 617.803,Z 1076.854,A -85,B 0,C 180,E1 27599.673,E2 27599.673} C_VEL
LIN {X 0,Y 619.889,Z 1059.056,A -85,B 0,C 180,E1 27597.95,E2 27597.95} C_VEL
LIN {X 0,Y 621.966,Z 1041.618,A -85,B 0,C 180,E1 27596.427,E2 27596.427} C_VEL
LIN {X 0,Y 624.674,Z 1019.548,A -85,B 0,C 180,E1 27594.703,E2 27594.703} C_VEL
LIN {X 0,Y 627.36,Z 996.425,A -85,B 0,C 180,E1 27593.139,E2 27593.139} C_VEL
LIN {X 0,Y 629.49,Z 977.555,A -85,B 0,C 180,E1 27592.007,E2 27592.007} C_VEL
LIN {X 0,Y 631.514,Z 958.702,A -85,B 0,C 180,E1 27590.998,E2 27590.998} C_VEL
LIN {X 0,Y 633.556,Z 938.34,A -85,B 0,C 180,E1 27590.036,E2 27590.036} C_VEL
LIN {X 0,Y 635.905,Z 913.021,A -85,B 0,C 180,E1 27589.004,E2 27589.004} C_VEL
LIN {X 0,Y 637.949,Z 886.565,A -85,B 0,C 180,E1 27588.131,E2 27588.131} C_VEL
LIN {X 0,Y 639.426,Z 864.549,A -85,B 0,C 180,E1 27587.541,E2 27587.541} C_VEL
LIN {X 0,Y 640.643,Z 842.48,A -85,B 0,C 180,E1 27587.068,E2 27587.068} C_VEL
LIN {X 0,Y 641.746,Z 815.019,A -85,B 0,C 180,E1 27586.629,E2 27586.629} C_VEL
LIN {X 0,Y 646.484,Z 591.916,A -85,B 0,C 180,E1 27583.613,E2 27583.613} C_VEL
LIN {X 0,Y 650.823,Z 401.097,A -85,B 0,C 180,E1 27580.961,E2 27580.961} C_VEL
LIN {X 0,Y 639.642,Z 384.575,A -85,B 0,C 180,E1 27579.511,E2 27579.511} C_VEL
LIN {X 0,Y 630.816,Z 371.716,A -85,B 0,C 180,E1 27578.27,E2 27578.27} C_VEL
LIN {X 0,Y 623.614,Z 361.699,A -85,B 0,C 180,E1 27577.191,E2 27577.191} C_VEL
LIN {X 0,Y 615.627,Z 351.204,A -85,B 0,C 180,E1 27575.926,E2 27575.926} C_VEL
LIN {X 0,Y 614.253,Z 349.025,A -85,B 0,C 180,E1 27575.645,E2 27575.645} C_VEL
LIN {X 0,Y 611.574,Z 343.595,A -85,B 0,C 180,E1 27574.678,E2 27574.678} C_VEL
LIN {X 0,Y 609.219,Z 339.338,A -85,B 0,C 180,E1 27573.855,E2 27573.855} C_VEL
LIN {X 0,Y 609.02,Z 338.364,A -85,B 0,C 180,E1 27573.706,E2 27573.706} C_VEL
LIN {X 0,Y 609.013,Z 338.335,A -85,B 0,C 180,E1 27570.836,E2 27570.836} C_VEL
LIN {X 0,Y 609.021,Z 338.334,A -85,B 0,C 180,E1 27567.558,E2 27567.558} C_VEL
LIN {X 0,Y 609.019,Z 338.368,A -85,B 0,C 180,E1 27564.647,E2 27564.647} C_VEL
LIN {X 0,Y 609.024,Z 338.342,A -85,B 0,C 180,E1 27561.376,E2 27561.376} C_VEL
LIN {X 0,Y 609.012,Z 338.348,A -85,B 0,C 180,E1 27558.573,E2 27558.573} C_VEL
LIN {X 0,Y 609.041,Z 338.363,A -85,B 0,C 180,E1 27555.327,E2 27555.327} C_VEL
LIN {X 0,Y 609.009,Z 338.33,A -85,B 0,C 180,E1 27552.42,E2 27552.42} C_VEL
LIN {X 0,Y 609.055,Z 338.365,A -85,B 0,C 180,E1 27549.258,E2 27549.258} C_VEL
LIN {X 0,Y 609.008,Z 338.332,A -85,B 0,C 180,E1 27546.316,E2 27546.316} C_VEL
LIN {X 0,Y 609.066,Z 338.355,A -85,B 0,C 180,E1 27543.2,E2 27543.2} C_VEL
LIN {X 0,Y 609.01,Z 338.344,A -85,B 0,C 180,E1 27540.188,E2 27540.188} C_VEL
LIN {X 0,Y 609.07,Z 338.339,A -85,B 0,C 180,E1 27537.078,E2 27537.078} C_VEL
LIN {X 0,Y 609.012,Z 338.361,A -85,B 0,C 180,E1 27534.063,E2 27534.063} C_VEL
LIN {X 0,Y 609.075,Z 338.328,A -85,B 0,C 180,E1 27531.028,E2 27531.028} C_VEL
LIN {X 0,Y 609.015,Z 338.368,A -85,B 0,C 180,E1 27527.965,E2 27527.965} C_VEL
LIN {X 0,Y 609.077,Z 338.325,A -85,B 0,C 180,E1 27524.852,E2 27524.852} C_VEL
LIN {X 0,Y 609.016,Z 338.351,A -85,B 0,C 180,E1 27521.823,E2 27521.823} C_VEL
LIN {X 0,Y 609.082,Z 338.359,A -85,B 0,C 180,E1 27518.728,E2 27518.728} C_VEL
LIN {X 0,Y 609.014,Z 338.339,A -85,B 0,C 180,E1 27515.663,E2 27515.663} C_VEL
LIN {X 0,Y 609.077,Z 338.359,A -85,B 0,C 180,E1 27512.635,E2 27512.635} C_VEL
LIN {X 0,Y 609.098,Z 338.5,A -85,B 0,C 180,E1 27512.397,E2 27512.397} C_VEL
LIN {X 0,Y 610.49,Z 342.076,A -85,B 0,C 180,E1 27511.782,E2 27511.782} C_VEL
LIN {X 0,Y 612.702,Z 344.868,A -85,B 0,C 180,E1 27511.408,E2 27511.408} C_VEL
LIN {X 0,Y 616.788,Z 349.854,A -85,B 0,C 180,E1 27510.74,E2 27510.74} C_VEL
LIN {X 0,Y 626.054,Z 362.128,A -85,B 0,C 180,E1 27509.29,E2 27509.29} C_VEL
LIN {X 0,Y 637.837,Z 378.646,A -85,B 0,C 180,E1 27507.593,E2 27507.593} C_VEL
LIN {X 0,Y 649.552,Z 395.947,A -85,B 0,C 180,E1 27506.055,E2 27506.055} C_VEL
LIN {X 0,Y 650.743,Z 398.194,A -85,B 0,C 180,E1 27505.896,E2 27505.896} C_VEL
LIN {X 0,Y 646.744,Z 571.43,A -85,B 0,C 180,E1 27503.488,E2 27503.488} C_VEL
LIN {X 0,Y 645.894,Z 579.135,A -85,B 0,C 180,E1 27503.446,E2 27503.446} C_VEL
LIN {X 0,Y 641.066,Z 599.791,A -85,B 0,C 180,E1 27503.571,E2 27503.571} C_VEL
LIN {X 0,Y 640.416,Z 606.398,A -85,B 0,C 180,E1 27503.527,E2 27503.527} C_VEL
LIN {X 0,Y 635.514,Z 817.002,A -85,B 0,C 180,E1 27500.646,E2 27500.646} C_VEL
LIN {X 0,Y 634.069,Z 845.791,A -85,B 0,C 180,E1 27500.111,E2 27500.111} C_VEL
LIN {X 0,Y 632.471,Z 869.37,A -85,B 0,C 180,E1 27499.521,E2 27499.521} C_VEL
LIN {X 0,Y 630.804,Z 890.669,A -85,B 0,C 180,E1 27498.866,E2 27498.866} C_VEL
LIN {X 0,Y 628.623,Z 915.32,A -85,B 0,C 180,E1 27497.96,E2 27497.96} C_VEL
LIN {X 0,Y 626.095,Z 939.875,A -85,B 0,C 180,E1 27496.871,E2 27496.871} C_VEL
LIN {X 0,Y 623.715,Z 961.245,A -85,B 0,C 180,E1 27495.772,E2 27495.772} C_VEL
LIN {X 0,Y 620.992,Z 984.677,A -85,B 0,C 180,E1 27494.394,E2 27494.394} C_VEL
LIN {X 0,Y 618.059,Z 1008.04,A -85,B 0,C 180,E1 27492.801,E2 27492.801} C_VEL
LIN {X 0,Y 615.327,Z 1029.319,A -85,B 0,C 180,E1 27491.154,E2 27491.154} C_VEL
LIN {X 0,Y 612.45,Z 1052.015,A -85,B 0,C 180,E1 27489.15,E2 27489.15} C_VEL
LIN {X 0,Y 609.982,Z 1071.544,A -85,B 0,C 180,E1 27487.188,E2 27487.188} C_VEL
LIN {X 0,Y 607.612,Z 1091.15,A -85,B 0,C 180,E1 27484.964,E2 27484.964} C_VEL
LIN {X 0,Y 605.568,Z 1109.056,A -85,B 0,C 180,E1 27482.638,E2 27482.638} C_VEL
LIN {X 0,Y 603.89,Z 1125.446,A -85,B 0,C 180,E1 27480.221,E2 27480.221} C_VEL
LIN {X 0,Y 602.575,Z 1139.765,A -85,B 0,C 180,E1 27477.792,E2 27477.792} C_VEL
LIN {X 0,Y 601.601,Z 1152.133,A -85,B 0,C 180,E1 27475.391,E2 27475.391} C_VEL
LIN {X 0,Y 600.89,Z 1163.054,A -85,B 0,C 180,E1 27472.915,E2 27472.915} C_VEL
LIN {X 0,Y 600.434,Z 1172.193,A -85,B 0,C 180,E1 27470.469,E2 27470.469} C_VEL
LIN {X 0,Y 600.135,Z 1180.251,A -85,B 0,C 180,E1 27467.852,E2 27467.852} C_VEL
LIN {X 0,Y 599.998,Z 1185.976,A -85,B 0,C 180,E1 27465.464,E2 27465.464} C_VEL
LIN {X 0,Y 599.932,Z 1190.289,A -85,B 0,C 180,E1 27463.1,E2 27463.1} C_VEL
LIN {X 0,Y 599.916,Z 1193.377,A -85,B 0,C 180,E1 27460.564,E2 27460.564} C_VEL
LIN {X 0,Y 599.909,Z 1194.73,A -85,B 0,C 180,E1 27458.144,E2 27458.144} C_VEL
LIN {X 0,Y 599.914,Z 1194.814,A -85,B 0,C 180,E1 27456.123,E2 27456.123} C_VEL
LIN {X 0,Y 599.911,Z 1193.879,A -85,B 0,C 180,E1 27454.014,E2 27454.014} C_VEL
LIN {X 0,Y 599.921,Z 1191.343,A -85,B 0,C 180,E1 27451.528,E2 27451.528} C_VEL
LIN {X 0,Y 599.983,Z 1187.024,A -85,B 0,C 180,E1 27448.95,E2 27448.95} C_VEL
LIN {X 0,Y 600.092,Z 1181.78,A -85,B 0,C 180,E1 27446.657,E2 27446.657} C_VEL
LIN {X 0,Y 600.319,Z 1174.946,A -85,B 0,C 180,E1 27444.265,E2 27444.265} C_VEL
LIN {X 0,Y 600.754,Z 1165.382,A -85,B 0,C 180,E1 27441.578,E2 27441.578} C_VEL
LIN {X 0,Y 601.403,Z 1155.17,A -85,B 0,C 180,E1 27439.172,E2 27439.172} C_VEL
LIN {X 0,Y 602.364,Z 1142.227,A -85,B 0,C 180,E1 27436.563,E2 27436.563} C_VEL
LIN {X 0,Y 603.67,Z 1127.625,A -85,B 0,C 180,E1 27434.041,E2 27434.041} C_VEL
LIN {X 0,Y 605.379,Z 1110.812,A -85,B 0,C 180,E1 27431.512,E2 27431.512} C_VEL
LIN {X 0,Y 607.316,Z 1093.615,A -85,B 0,C 180,E1 27429.255,E2 27429.255} C_VEL
LIN {X 0,Y 609.63,Z 1074.402,A -85,B 0,C 180,E1 27427.024,E2 27427.024} C_VEL
LIN {X 0,Y 612.049,Z 1055.054,A -85,B 0,C 180,E1 27425.053,E2 27425.053} C_VEL
LIN {X 0,Y 614.712,Z 1034.304,A -85,B 0,C 180,E1 27423.169,E2 27423.169} C_VEL
LIN {X 0,Y 617.505,Z 1012.207,A -85,B 0,C 180,E1 27421.415,E2 27421.415} C_VEL
LIN {X 0,Y 620.223,Z 990.724,A -85,B 0,C 180,E1 27419.91,E2 27419.91} C_VEL
LIN {X 0,Y 623.194,Z 966.161,A -85,B 0,C 180,E1 27418.41,E2 27418.41} C_VEL
LIN {X 0,Y 625.644,Z 944.166,A -85,B 0,C 180,E1 27417.251,E2 27417.251} C_VEL
LIN {X 0,Y 627.72,Z 924.369,A -85,B 0,C 180,E1 27416.337,E2 27416.337} C_VEL
LIN {X 0,Y 629.872,Z 901.618,A -85,B 0,C 180,E1 27415.424,E2 27415.424} C_VEL
LIN {X 0,Y 632.144,Z 874.195,A -85,B 0,C 180,E1 27414.527,E2 27414.527} C_VEL
LIN {X 0,Y 633.676,Z 851.844,A -85,B 0,C 180,E1 27413.939,E2 27413.939} C_VEL
LIN {X 0,Y 634.903,Z 829.966,A -85,B 0,C 180,E1 27413.481,E2 27413.481} C_VEL
LIN {X 0,Y 636.006,Z 801.709,A -85,B 0,C 180,E1 27413.042,E2 27413.042} C_VEL
LIN {X 0,Y 641.044,Z 579.738,A -85,B 0,C 180,E1 27410.015,E2 27410.015} C_VEL
LIN {X 0,Y 645.353,Z 401.676,A -85,B 0,C 180,E1 27407.519,E2 27407.519} C_VEL
LIN {X 0,Y 636.453,Z 388.461,A -85,B 0,C 180,E1 27406.341,E2 27406.341} C_VEL
LIN {X 0,Y 625.829,Z 373.528,A -85,B 0,C 180,E1 27404.893,E2 27404.893} C_VEL
LIN {X 0,Y 611.111,Z 353.957,A -85,B 0,C 180,E1 27402.799,E2 27402.799} C_VEL
LIN {X 0,Y 603.54,Z 344.127,A -85,B 0,C 180,E1 27401.661,E2 27401.661} C_VEL
LIN {X 0,Y 601.605,Z 341.373,A -85,B 0,C 180,E1 27401.304,E2 27401.304} C_VEL
LIN {X 0,Y 601.047,Z 339.344,A -85,B 0,C 180,E1 27400.997,E2 27400.997} C_VEL
LIN {X 0,Y 601.049,Z 339.364,A -85,B 0,C 180,E1 27398.263,E2 27398.263} C_VEL
LIN {X 0,Y 601.055,Z 339.352,A -85,B 0,C 180,E1 27394.905,E2 27394.905} C_VEL
LIN {X 0,Y 601.049,Z 339.353,A -85,B 0,C 180,E1 27392.142,E2 27392.142} C_VEL
LIN {X 0,Y 601.074,Z 339.324,A -85,B 0,C 180,E1 27388.952,E2 27388.952} C_VEL
LIN {X 0,Y 601.043,Z 339.345,A -85,B 0,C 180,E1 27386.158,E2 27386.158} C_VEL
LIN {X 0,Y 601.117,Z 339.323,A -85,B 0,C 180,E1 27383.1,E2 27383.1} C_VEL
LIN {X 0,Y 601.04,Z 339.336,A -85,B 0,C 180,E1 27380.143,E2 27380.143} C_VEL
LIN {X 0,Y 601.119,Z 339.344,A -85,B 0,C 180,E1 27377.123,E2 27377.123} C_VEL
LIN {X 0,Y 601.045,Z 339.355,A -85,B 0,C 180,E1 27374.057,E2 27374.057} C_VEL
LIN {X 0,Y 601.105,Z 339.355,A -85,B 0,C 180,E1 27371.073,E2 27371.073} C_VEL
LIN {X 0,Y 601.048,Z 339.359,A -85,B 0,C 180,E1 27367.937,E2 27367.937} C_VEL
LIN {X 0,Y 601.078,Z 339.35,A -85,B 0,C 180,E1 27365.154,E2 27365.154} C_VEL
LIN {X 0,Y 601.055,Z 339.354,A -85,B 0,C 180,E1 27361.907,E2 27361.907} C_VEL
LIN {X 0,Y 601.059,Z 339.349,A -85,B 0,C 180,E1 27359.237,E2 27359.237} C_VEL
LIN {X 0,Y 601.065,Z 339.345,A -85,B 0,C 180,E1 27355.898,E2 27355.898} C_VEL
LIN {X 0,Y 601.058,Z 339.359,A -85,B 0,C 180,E1 27353.121,E2 27353.121} C_VEL
LIN {X 0,Y 601.078,Z 339.353,A -85,B 0,C 180,E1 27349.844,E2 27349.844} C_VEL
LIN {X 0,Y 601.051,Z 339.308,A -85,B 0,C 180,E1 27347.022,E2 27347.022} C_VEL
LIN {X 0,Y 601.104,Z 339.355,A -85,B 0,C 180,E1 27343.871,E2 27343.871} C_VEL
LIN {X 0,Y 601.051,Z 339.311,A -85,B 0,C 180,E1 27340.97,E2 27340.97} C_VEL
LIN {X 0,Y 601.119,Z 339.353,A -85,B 0,C 180,E1 27337.816,E2 27337.816} C_VEL
LIN {X 0,Y 601.053,Z 339.313,A -85,B 0,C 180,E1 27334.794,E2 27334.794} C_VEL
LIN {X 0,Y 601.117,Z 339.344,A -85,B 0,C 180,E1 27331.63,E2 27331.63} C_VEL
LIN {X 0,Y 601.058,Z 339.352,A -85,B 0,C 180,E1 27328.733,E2 27328.733} C_VEL
LIN {X 0,Y 601.07,Z 339.446,A -85,B 0,C 180,E1 27326.704,E2 27326.704} C_VEL
LIN {X 0,Y 602.276,Z 342.668,A -85,B 0,C 180,E1 27326.209,E2 27326.209} C_VEL
LIN {X 0,Y 603.573,Z 344.676,A -85,B 0,C 180,E1 27325.834,E2 27325.834} C_VEL
LIN {X 0,Y 606.164,Z 350.023,A -85,B 0,C 180,E1 27324.996,E2 27324.996} C_VEL
LIN {X 0,Y 621.573,Z 370.687,A -85,B 0,C 180,E1 27322.753,E2 27322.753} C_VEL
LIN {X 0,Y 634.275,Z 388.362,A -85,B 0,C 180,E1 27321.009,E2 27321.009} C_VEL
LIN {X 0,Y 645.501,Z 405.116,A -85,B 0,C 180,E1 27319.518,E2 27319.518} C_VEL
LIN {X 0,Y 640.557,Z 608.969,A -85,B 0,C 180,E1 27316.672,E2 27316.672} C_VEL
LIN {X 0,Y 635.609,Z 823.764,A -85,B 0,C 180,E1 27313.738,E2 27313.738} C_VEL
LIN {X 0,Y 634.61,Z 845.646,A -85,B 0,C 180,E1 27313.365,E2 27313.365} C_VEL
LIN {X 0,Y 633.307,Z 867.513,A -85,B 0,C 180,E1 27312.879,E2 27312.879} C_VEL
LIN {X 0,Y 631.438,Z 893.753,A -85,B 0,C 180,E1 27312.143,E2 27312.143} C_VEL
LIN {X 0,Y 629.207,Z 918.734,A -85,B 0,C 180,E1 27311.259,E2 27311.259} C_VEL
LIN {X 0,Y 627.184,Z 939.464,A -85,B 0,C 180,E1 27310.394,E2 27310.394} C_VEL
LIN {X 0,Y 625.147,Z 958.693,A -85,B 0,C 180,E1 27309.476,E2 27309.476} C_VEL
LIN {X 0,Y 622.956,Z 977.949,A -85,B 0,C 180,E1 27308.438,E2 27308.438} C_VEL
LIN {X 0,Y 620.584,Z 997.794,A -85,B 0,C 180,E1 27307.234,E2 27307.234} C_VEL
LIN {X 0,Y 617.515,Z 1022.228,A -85,B 0,C 180,E1 27305.54,E2 27305.54} C_VEL
LIN {X 0,Y 614.968,Z 1041.905,A -85,B 0,C 180,E1 27303.981,E2 27303.981} C_VEL
LIN {X 0,Y 612.783,Z 1059.055,A -85,B 0,C 180,E1 27302.467,E2 27302.467} C_VEL
LIN {X 0,Y 610.531,Z 1077.072,A -85,B 0,C 180,E1 27300.704,E2 27300.704} C_VEL
LIN {X 0,Y 608.059,Z 1097.15,A -85,B 0,C 180,E1 27298.48,E2 27298.48} C_VEL
LIN {X 0,Y 606.258,Z 1112.619,A -85,B 0,C 180,E1 27296.547,E2 27296.547} C_VEL
LIN {X 0,Y 604.64,Z 1127.891,A -85,B 0,C 180,E1 27294.419,E2 27294.419} C_VEL
LIN {X 0,Y 603.101,Z 1143.702,A -85,B 0,C 180,E1 27291.902,E2 27291.902} C_VEL
LIN {X 0,Y 602.121,Z 1155.273,A -85,B 0,C 180,E1 27289.801,E2 27289.801} C_VEL
LIN {X 0,Y 601.343,Z 1165.909,A -85,B 0,C 180,E1 27287.615,E2 27287.615} C_VEL
LIN {X 0,Y 600.69,Z 1177.02,A -85,B 0,C 180,E1 27284.951,E2 27284.951} C_VEL
LIN {X 0,Y 600.299,Z 1185.324,A -85,B 0,C 180,E1 27282.557,E2 27282.557} C_VEL
LIN {X 0,Y 600.092,Z 1191.863,A -85,B 0,C 180,E1 27280.27,E2 27280.27} C_VEL
LIN {X 0,Y 599.973,Z 1197.543,A -85,B 0,C 180,E1 27277.758,E2 27277.758} C_VEL
LIN {X 0,Y 599.926,Z 1201.663,A -85,B 0,C 180,E1 27275.163,E2 27275.163} C_VEL
LIN {X 0,Y 599.915,Z 1203.927,A -85,B 0,C 180,E1 27272.866,E2 27272.866} C_VEL
LIN {X 0,Y 599.895,Z 1204.849,A -85,B 0,C 180,E1 27270.668,E2 27270.668} C_VEL
LIN {X 0,Y 599.908,Z 1204.623,A -85,B 0,C 180,E1 27268.376,E2 27268.376} C_VEL
LIN {X 0,Y 599.918,Z 1202.789,A -85,B 0,C 180,E1 27265.795,E2 27265.795} C_VEL
LIN {X 0,Y 599.944,Z 1199.513,A -85,B 0,C 180,E1 27263.375,E2 27263.375} C_VEL
LIN {X 0,Y 600.014,Z 1195.105,A -85,B 0,C 180,E1 27261.085,E2 27261.085} C_VEL
LIN {X 0,Y 600.197,Z 1188.476,A -85,B 0,C 180,E1 27258.469,E2 27258.469} C_VEL
LIN {X 0,Y 600.505,Z 1180.572,A -85,B 0,C 180,E1 27256.029,E2 27256.029} C_VEL
LIN {X 0,Y 600.938,Z 1172.306,A -85,B 0,C 180,E1 27253.868,E2 27253.868} C_VEL
LIN {X 0,Y 601.566,Z 1162.692,A -85,B 0,C 180,E1 27251.691,E2 27251.691} C_VEL
LIN {X 0,Y 602.621,Z 1149.398,A -85,B 0,C 180,E1 27249.092,E2 27249.092} C_VEL
LIN {X 0,Y 603.844,Z 1135.741,A -85,B 0,C 180,E1 27246.791,E2 27246.791} C_VEL
LIN {X 0,Y 605.279,Z 1121.578,A -85,B 0,C 180,E1 27244.669,E2 27244.669} C_VEL
LIN {X 0,Y 607.376,Z 1103.066,A -85,B 0,C 180,E1 27242.233,E2 27242.233} C_VEL
LIN {X 0,Y 609.273,Z 1086.965,A -85,B 0,C 180,E1 27240.359,E2 27240.359} C_VEL
LIN {X 0,Y 611.356,Z 1070.397,A -85,B 0,C 180,E1 27238.622,E2 27238.622} C_VEL
LIN {X 0,Y 614.09,Z 1049.297,A -85,B 0,C 180,E1 27236.647,E2 27236.647} C_VEL
LIN {X 0,Y 616.657,Z 1028.87,A -85,B 0,C 180,E1 27234.969,E2 27234.969} C_VEL
LIN {X 0,Y 619.038,Z 1009.977,A -85,B 0,C 180,E1 27233.583,E2 27233.583} C_VEL
LIN {X 0,Y 621.631,Z 988.944,A -85,B 0,C 180,E1 27232.207,E2 27232.207} C_VEL
LIN {X 0,Y 624.587,Z 963.722,A -85,B 0,C 180,E1 27230.778,E2 27230.778} C_VEL
LIN {X 0,Y 626.818,Z 942.858,A -85,B 0,C 180,E1 27229.757,E2 27229.757} C_VEL
LIN {X 0,Y 628.829,Z 922.587,A -85,B 0,C 180,E1 27228.892,E2 27228.892} C_VEL
LIN {X 0,Y 630.688,Z 901.904,A -85,B 0,C 180,E1 27228.131,E2 27228.131} C_VEL
LIN {X 0,Y 632.495,Z 879.261,A -85,B 0,C 180,E1 27227.429,E2 27227.429} C_VEL
LIN {X 0,Y 634.363,Z 850.616,A -85,B 0,C 180,E1 27226.733,E2 27226.733} C_VEL
LIN {X 0,Y 635.496,Z 826.763,A -85,B 0,C 180,E1 27226.307,E2 27226.307} C_VEL
LIN {X 0,Y 639.957,Z 634.726,A -85,B 0,C 180,E1 27223.684,E2 27223.684} C_VEL
LIN {X 0,Y 644.968,Z 426.413,A -85,B 0,C 180,E1 27220.784,E2 27220.784} C_VEL
LIN {X 0,Y 645.373,Z 404.806,A -85,B 0,C 180,E1 27220.464,E2 27220.464} C_VEL
LIN {X 0,Y 630.084,Z 381.938,A -85,B 0,C 180,E1 27218.372,E2 27218.372} C_VEL
LIN {X 0,Y 620.224,Z 368.12,A -85,B 0,C 180,E1 27216.879,E2 27216.879} C_VEL
LIN {X 0,Y 609.896,Z 354.355,A -85,B 0,C 180,E1 27215.188,E2 27215.188} C_VEL
LIN {X 0,Y 606.523,Z 350.044,A -85,B 0,C 180,E1 27214.606,E2 27214.606} C_VEL
LIN {X 0,Y 605.688,Z 348.531,A -85,B 0,C 180,E1 27214.372,E2 27214.372} C_VEL
LIN {X 0,Y 603.826,Z 345.024,A -85,B 0,C 180,E1 27213.693,E2 27213.693} C_VEL
LIN {X 0,Y 602.671,Z 343.257,A -85,B 0,C 180,E1 27213.31,E2 27213.31} C_VEL
LIN {X 0,Y 601.213,Z 340.044,A -85,B 0,C 180,E1 27212.7,E2 27212.7} C_VEL
LIN {X 0,Y 601.108,Z 339.334,A -85,B 0,C 180,E1 27212.555,E2 27212.555} C_VEL
LIN {X 0,Y 601.073,Z 339.358,A -85,B 0,C 180,E1 27209.389,E2 27209.389} C_VEL
LIN {X 0,Y 601.096,Z 339.319,A -85,B 0,C 180,E1 27206.475,E2 27206.475} C_VEL
LIN {X 0,Y 601.078,Z 339.329,A -85,B 0,C 180,E1 27203.323,E2 27203.323} C_VEL
LIN {X 0,Y 601.087,Z 339.352,A -85,B 0,C 180,E1 27200.446,E2 27200.446} C_VEL
LIN {X 0,Y 601.075,Z 339.32,A -85,B 0,C 180,E1 27197.124,E2 27197.124} C_VEL
LIN {X 0,Y 601.089,Z 339.356,A -85,B 0,C 180,E1 27194.252,E2 27194.252} C_VEL
LIN {X 0,Y 601.078,Z 339.333,A -85,B 0,C 180,E1 27190.932,E2 27190.932} C_VEL
LIN {X 0,Y 601.092,Z 339.333,A -85,B 0,C 180,E1 27188.032,E2 27188.032} C_VEL
LIN {X 0,Y 601.083,Z 339.35,A -85,B 0,C 180,E1 27184.771,E2 27184.771} C_VEL
LIN {X 0,Y 601.096,Z 339.319,A -85,B 0,C 180,E1 27181.811,E2 27181.811} C_VEL
LIN {X 0,Y 601.083,Z 339.358,A -85,B 0,C 180,E1 27178.57,E2 27178.57} C_VEL
LIN {X 0,Y 601.099,Z 339.312,A -85,B 0,C 180,E1 27175.612,E2 27175.612} C_VEL
LIN {X 0,Y 601.082,Z 339.35,A -85,B 0,C 180,E1 27172.352,E2 27172.352} C_VEL
LIN {X 0,Y 601.109,Z 339.326,A -85,B 0,C 180,E1 27169.36,E2 27169.36} C_VEL
LIN {X 0,Y 601.077,Z 339.324,A -85,B 0,C 180,E1 27166.14,E2 27166.14} C_VEL
LIN {X 0,Y 601.115,Z 339.351,A -85,B 0,C 180,E1 27163.176,E2 27163.176} C_VEL
LIN {X 0,Y 601.081,Z 339.325,A -85,B 0,C 180,E1 27159.96,E2 27159.96} C_VEL
LIN {X 0,Y 601.114,Z 339.324,A -85,B 0,C 180,E1 27156.989,E2 27156.989} C_VEL
LIN {X 0,Y 601.085,Z 339.353,A -85,B 0,C 180,E1 27153.737,E2 27153.737} C_VEL
LIN {X 0,Y 601.095,Z 339.452,A -85,B 0,C 180,E1 27153.525,E2 27153.525} C_VEL
LIN {X 0,Y 602.379,Z 342.78,A -85,B 0,C 180,E1 27152.974,E2 27152.974} C_VEL
LIN {X 0,Y 605.101,Z 345.828,A -85,B 0,C 180,E1 27152.493,E2 27152.493} C_VEL
LIN {X 0,Y 610.104,Z 352.258,A -85,B 0,C 180,E1 27151.622,E2 27151.622} C_VEL
LIN {X 0,Y 613.785,Z 356.766,A -85,B 0,C 180,E1 27151.011,E2 27151.011} C_VEL
LIN {X 0,Y 624.517,Z 371.019,A -85,B 0,C 180,E1 27149.313,E2 27149.313} C_VEL
LIN {X 0,Y 635.409,Z 386.858,A -85,B 0,C 180,E1 27147.721,E2 27147.721} C_VEL
LIN {X 0,Y 645.362,Z 401.599,A -85,B 0,C 180,E1 27146.392,E2 27146.392} C_VEL
LIN {X 0,Y 640.984,Z 582.235,A -85,B 0,C 180,E1 27143.86,E2 27143.86} C_VEL
LIN {X 0,Y 640.416,Z 606.398,A -85,B 0,C 180,E1 27143.527,E2 27143.527} C_VEL
LIN {X 0,Y 639.581,Z 614.099,A -85,B 0,C 180,E1 27143.483,E2 27143.483} C_VEL
LIN {X 0,Y 634.75,Z 634.752,A -85,B 0,C 180,E1 27143.61,E2 27143.61} C_VEL
LIN {X 0,Y 634.057,Z 641.365,A -85,B 0,C 180,E1 27143.569,E2 27143.569} C_VEL
LIN {X 0,Y 629.668,Z 818.669,A -85,B 0,C 180,E1 27141.126,E2 27141.126} C_VEL
LIN {X 0,Y 628.115,Z 847.246,A -85,B 0,C 180,E1 27140.58,E2 27140.58} C_VEL
LIN {X 0,Y 626.5,Z 869.798,A -85,B 0,C 180,E1 27140.009,E2 27140.009} C_VEL
LIN {X 0,Y 624.73,Z 891.288,A -85,B 0,C 180,E1 27139.342,E2 27139.342} C_VEL
LIN {X 0,Y 622.308,Z 917.156,A -85,B 0,C 180,E1 27138.379,E2 27138.379} C_VEL
LIN {X 0,Y 619.697,Z 940.886,A -85,B 0,C 180,E1 27137.308,E2 27137.308} C_VEL
LIN {X 0,Y 617.197,Z 962.142,A -85,B 0,C 180,E1 27136.202,E2 27136.202} C_VEL
LIN {X 0,Y 614.22,Z 986.316,A -85,B 0,C 180,E1 27134.759,E2 27134.759} C_VEL
LIN {X 0,Y 611.224,Z 1008.764,A -85,B 0,C 180,E1 27133.204,E2 27133.204} C_VEL
LIN {X 0,Y 608.439,Z 1029.297,A -85,B 0,C 180,E1 27131.598,E2 27131.598} C_VEL
LIN {X 0,Y 605.399,Z 1051.685,A -85,B 0,C 180,E1 27129.606,E2 27129.606} C_VEL
LIN {X 0,Y 602.882,Z 1070.412,A -85,B 0,C 180,E1 27127.71,E2 27127.71} C_VEL
LIN {X 0,Y 600.452,Z 1089.096,A -85,B 0,C 180,E1 27125.59,E2 27125.59} C_VEL
LIN {X 0,Y 598.316,Z 1106.617,A -85,B 0,C 180,E1 27123.322,E2 27123.322} C_VEL
LIN {X 0,Y 596.578,Z 1122.026,A -85,B 0,C 180,E1 27121.078,E2 27121.078} C_VEL
LIN {X 0,Y 595.021,Z 1137.484,A -85,B 0,C 180,E1 27118.494,E2 27118.494} C_VEL
LIN {X 0,Y 593.874,Z 1150.629,A -85,B 0,C 180,E1 27115.96,E2 27115.96} C_VEL
LIN {X 0,Y 593.019,Z 1162.673,A -85,B 0,C 180,E1 27113.23,E2 27113.23} C_VEL
LIN {X 0,Y 592.498,Z 1171.742,A -85,B 0,C 180,E1 27110.784,E2 27110.784} C_VEL
LIN {X 0,Y 592.18,Z 1179.426,A -85,B 0,C 180,E1 27108.303,E2 27108.303} C_VEL
LIN {X 0,Y 592.016,Z 1185.734,A -85,B 0,C 180,E1 27105.696,E2 27105.696} C_VEL
LIN {X 0,Y 591.942,Z 1190.017,A -85,B 0,C 180,E1 27103.353,E2 27103.353} C_VEL
LIN {X 0,Y 591.912,Z 1193.212,A -85,B 0,C 180,E1 27100.807,E2 27100.807} C_VEL
LIN {X 0,Y 591.915,Z 1194.686,A -85,B 0,C 180,E1 27098.353,E2 27098.353} C_VEL
LIN {X 0,Y 591.913,Z 1194.836,A -85,B 0,C 180,E1 27096.206,E2 27096.206} C_VEL
LIN {X 0,Y 591.912,Z 1193.941,A -85,B 0,C 180,E1 27094.068,E2 27094.068} C_VEL
LIN {X 0,Y 591.921,Z 1191.589,A -85,B 0,C 180,E1 27091.646,E2 27091.646} C_VEL
LIN {X 0,Y 591.983,Z 1187.406,A -85,B 0,C 180,E1 27089.032,E2 27089.032} C_VEL
LIN {X 0,Y 592.1,Z 1182.017,A -85,B 0,C 180,E1 27086.612,E2 27086.612} C_VEL
LIN {X 0,Y 592.33,Z 1175.518,A -85,B 0,C 180,E1 27084.284,E2 27084.284} C_VEL
LIN {X 0,Y 592.788,Z 1166.145,A -85,B 0,C 180,E1 27081.562,E2 27081.562} C_VEL
LIN {X 0,Y 593.499,Z 1155.6,A -85,B 0,C 180,E1 27079.026,E2 27079.026} C_VEL
LIN {X 0,Y 594.493,Z 1143.083,A -85,B 0,C 180,E1 27076.448,E2 27076.448} C_VEL
LIN {X 0,Y 595.787,Z 1129.405,A -85,B 0,C 180,E1 27074.025,E2 27074.025} C_VEL
LIN {X 0,Y 597.457,Z 1113.897,A -85,B 0,C 180,E1 27071.609,E2 27071.609} C_VEL
LIN {X 0,Y 599.494,Z 1096.858,A -85,B 0,C 180,E1 27069.294,E2 27069.294} C_VEL
LIN {X 0,Y 601.762,Z 1078.837,A -85,B 0,C 180,E1 27067.12,E2 27067.12} C_VEL
LIN {X 0,Y 604.511,Z 1058.29,A -85,B 0,C 180,E1 27064.949,E2 27064.949} C_VEL
LIN {X 0,Y 607.157,Z 1038.777,A -85,B 0,C 180,E1 27063.125,E2 27063.125} C_VEL
LIN {X 0,Y 610.139,Z 1016.826,A -85,B 0,C 180,E1 27061.305,E2 27061.305} C_VEL
LIN {X 0,Y 613.024,Z 995.069,A -85,B 0,C 180,E1 27059.736,E2 27059.736} C_VEL
LIN {X 0,Y 615.806,Z 973.645,A -85,B 0,C 180,E1 27058.37,E2 27058.37} C_VEL
LIN {X 0,Y 618.906,Z 948.175,A -85,B 0,C 180,E1 27056.965,E2 27056.965} C_VEL
LIN {X 0,Y 621.173,Z 927.763,A -85,B 0,C 180,E1 27055.995,E2 27055.995} C_VEL
LIN {X 0,Y 623.174,Z 907.848,A -85,B 0,C 180,E1 27055.167,E2 27055.167} C_VEL
LIN {X 0,Y 625.186,Z 886.19,A -85,B 0,C 180,E1 27054.399,E2 27054.399} C_VEL
LIN {X 0,Y 627.31,Z 859.76,A -85,B 0,C 180,E1 27053.626,E2 27053.626} C_VEL
LIN {X 0,Y 628.862,Z 834.268,A -85,B 0,C 180,E1 27053.059,E2 27053.059} C_VEL
LIN {X 0,Y 629.959,Z 810.7,A -85,B 0,C 180,E1 27052.665,E2 27052.665} C_VEL
LIN {X 0,Y 635.273,Z 592.191,A -85,B 0,C 180,E1 27049.659,E2 27049.659} C_VEL
LIN {X 0,Y 640.081,Z 405.67,A -85,B 0,C 180,E1 27047.032,E2 27047.032} C_VEL
LIN {X 0,Y 628.761,Z 388.934,A -85,B 0,C 180,E1 27045.499,E2 27045.499} C_VEL
LIN {X 0,Y 615.709,Z 371.221,A -85,B 0,C 180,E1 27043.677,E2 27043.677} C_VEL
LIN {X 0,Y 607.222,Z 359.928,A -85,B 0,C 180,E1 27042.433,E2 27042.433} C_VEL
LIN {X 0,Y 599.852,Z 350.345,A -85,B 0,C 180,E1 27041.307,E2 27041.307} C_VEL
LIN {X 0,Y 596.432,Z 345.894,A -85,B 0,C 180,E1 27040.767,E2 27040.767} C_VEL
LIN {X 0,Y 594.05,Z 343.242,A -85,B 0,C 180,E1 27040.393,E2 27040.393} C_VEL
LIN {X 0,Y 593.339,Z 341.467,A -85,B 0,C 180,E1 27040.198,E2 27040.198} C_VEL
LIN {X 0,Y 593.139,Z 340.349,A -85,B 0,C 180,E1 27040.004,E2 27040.004} C_VEL
LIN {X 0,Y 593.105,Z 340.345,A -85,B 0,C 180,E1 27036.798,E2 27036.798} C_VEL
LIN {X 0,Y 593.132,Z 340.342,A -85,B 0,C 180,E1 27033.917,E2 27033.917} C_VEL
LIN {X 0,Y 593.114,Z 340.35,A -85,B 0,C 180,E1 27030.712,E2 27030.712} C_VEL
LIN {X 0,Y 593.109,Z 340.299,A -85,B 0,C 180,E1 27027.948,E2 27027.948} C_VEL
LIN {X 0,Y 593.118,Z 340.348,A -85,B 0,C 180,E1 27024.608,E2 27024.608} C_VEL
LIN {X 0,Y 593.114,Z 340.296,A -85,B 0,C 180,E1 27021.77,E2 27021.77} C_VEL
LIN {X 0,Y 593.122,Z 340.348,A -85,B 0,C 180,E1 27018.478,E2 27018.478} C_VEL
LIN {X 0,Y 593.117,Z 340.343,A -85,B 0,C 180,E1 27015.648,E2 27015.648} C_VEL
LIN {X 0,Y 593.118,Z 340.347,A -85,B 0,C 180,E1 27012.264,E2 27012.264} C_VEL
LIN {X 0,Y 593.124,Z 340.334,A -85,B 0,C 180,E1 27009.412,E2 27009.412} C_VEL
LIN {X 0,Y 593.119,Z 340.335,A -85,B 0,C 180,E1 27006.097,E2 27006.097} C_VEL
LIN {X 0,Y 593.123,Z 340.343,A -85,B 0,C 180,E1 27003.286,E2 27003.286} C_VEL
LIN {X 0,Y 593.126,Z 340.341,A -85,B 0,C 180,E1 27000,E2 27000} C_VEL
LIN {X 0,Y 593.121,Z 340.348,A -85,B 0,C 180,E1 26997.198,E2 26997.198} C_VEL
LIN {X 0,Y 593.133,Z 340.347,A -85,B 0,C 180,E1 26993.903,E2 26993.903} C_VEL
LIN {X 0,Y 593.121,Z 340.343,A -85,B 0,C 180,E1 26991.06,E2 26991.06} C_VEL
LIN {X 0,Y 593.139,Z 340.298,A -85,B 0,C 180,E1 26987.835,E2 26987.835} C_VEL
LIN {X 0,Y 593.117,Z 340.338,A -85,B 0,C 180,E1 26985.004,E2 26985.004} C_VEL
LIN {X 0,Y 593.161,Z 340.303,A -85,B 0,C 180,E1 26981.829,E2 26981.829} C_VEL
LIN {X 0,Y 593.118,Z 340.341,A -85,B 0,C 180,E1 26978.853,E2 26978.853} C_VEL
LIN {X 0,Y 593.174,Z 340.295,A -85,B 0,C 180,E1 26975.771,E2 26975.771} C_VEL
LIN {X 0,Y 593.123,Z 340.349,A -85,B 0,C 180,E1 26972.707,E2 26972.707} C_VEL
LIN {X 0,Y 593.184,Z 340.336,A -85,B 0,C 180,E1 26969.623,E2 26969.623} C_VEL
LIN {X 0,Y 593.213,Z 340.486,A -85,B 0,C 180,E1 26967.656,E2 26967.656} C_VEL
LIN {X 0,Y 594.546,Z 343.977,A -85,B 0,C 180,E1 26967.097,E2 26967.097} C_VEL
LIN {X 0,Y 595.524,Z 345.4,A -85,B 0,C 180,E1 26966.814,E2 26966.814} C_VEL
LIN {X 0,Y 597.17,Z 348.892,A -85,B 0,C 180,E1 26966.227,E2 26966.227} C_VEL
LIN {X 0,Y 598.368,Z 350.627,A -85,B 0,C 180,E1 26965.987,E2 26965.987} C_VEL
LIN {X 0,Y 613.766,Z 371.34,A -85,B 0,C 180,E1 26963.659,E2 26963.659} C_VEL
LIN {X 0,Y 627.869,Z 390.756,A -85,B 0,C 180,E1 26961.677,E2 26961.677} C_VEL
LIN {X 0,Y 640.194,Z 409.01,A -85,B 0,C 180,E1 26960.01,E2 26960.01} C_VEL
LIN {X 0,Y 634.99,Z 611.675,A -85,B 0,C 180,E1 26957.161,E2 26957.161} C_VEL
LIN {X 0,Y 629.798,Z 824.271,A -85,B 0,C 180,E1 26954.234,E2 26954.234} C_VEL
LIN {X 0,Y 628.751,Z 846.049,A -85,B 0,C 180,E1 26953.859,E2 26953.859} C_VEL
LIN {X 0,Y 627.369,Z 868.132,A -85,B 0,C 180,E1 26953.365,E2 26953.365} C_VEL
LIN {X 0,Y 625.39,Z 894.354,A -85,B 0,C 180,E1 26952.622,E2 26952.622} C_VEL
LIN {X 0,Y 623.048,Z 919.243,A -85,B 0,C 180,E1 26951.733,E2 26951.733} C_VEL
LIN {X 0,Y 620.977,Z 939.461,A -85,B 0,C 180,E1 26950.883,E2 26950.883} C_VEL
LIN {X 0,Y 618.823,Z 958.69,A -85,B 0,C 180,E1 26949.96,E2 26949.96} C_VEL
LIN {X 0,Y 616.543,Z 977.639,A -85,B 0,C 180,E1 26948.933,E2 26948.933} C_VEL
LIN {X 0,Y 614.088,Z 997.061,A -85,B 0,C 180,E1 26947.749,E2 26947.749} C_VEL
LIN {X 0,Y 610.965,Z 1020.891,A -85,B 0,C 180,E1 26946.096,E2 26946.096} C_VEL
LIN {X 0,Y 608.093,Z 1041.619,A -85,B 0,C 180,E1 26944.445,E2 26944.445} C_VEL
LIN {X 0,Y 605.719,Z 1059.054,A -85,B 0,C 180,E1 26942.893,E2 26942.893} C_VEL
LIN {X 0,Y 603.288,Z 1077.267,A -85,B 0,C 180,E1 26941.092,E2 26941.092} C_VEL
LIN {X 0,Y 600.702,Z 1097.148,A -85,B 0,C 180,E1 26938.862,E2 26938.862} C_VEL
LIN {X 0,Y 598.745,Z 1112.645,A -85,B 0,C 180,E1 26936.903,E2 26936.903} C_VEL
LIN {X 0,Y 597.074,Z 1127.45,A -85,B 0,C 180,E1 26934.815,E2 26934.815} C_VEL
LIN {X 0,Y 595.364,Z 1143.704,A -85,B 0,C 180,E1 26932.201,E2 26932.201} C_VEL
LIN {X 0,Y 594.298,Z 1155.271,A -85,B 0,C 180,E1 26930.073,E2 26930.073} C_VEL
LIN {X 0,Y 593.5,Z 1165.449,A -85,B 0,C 180,E1 26927.957,E2 26927.957} C_VEL
LIN {X 0,Y 592.788,Z 1176.306,A -85,B 0,C 180,E1 26925.356,E2 26925.356} C_VEL
LIN {X 0,Y 592.348,Z 1185.18,A -85,B 0,C 180,E1 26922.775,E2 26922.775} C_VEL
LIN {X 0,Y 592.108,Z 1191.86,A -85,B 0,C 180,E1 26920.41,E2 26920.41} C_VEL
LIN {X 0,Y 591.983,Z 1197.542,A -85,B 0,C 180,E1 26917.863,E2 26917.863} C_VEL
LIN {X 0,Y 591.927,Z 1201.661,A -85,B 0,C 180,E1 26915.233,E2 26915.233} C_VEL
LIN {X 0,Y 591.915,Z 1203.925,A -85,B 0,C 180,E1 26912.905,E2 26912.905} C_VEL
LIN {X 0,Y 591.895,Z 1204.849,A -85,B 0,C 180,E1 26910.678,E2 26910.678} C_VEL
LIN {X 0,Y 591.908,Z 1204.623,A -85,B 0,C 180,E1 26908.354,E2 26908.354} C_VEL
LIN {X 0,Y 591.918,Z 1202.789,A -85,B 0,C 180,E1 26905.738,E2 26905.738} C_VEL
LIN {X 0,Y 591.945,Z 1199.546,A -85,B 0,C 180,E1 26903.307,E2 26903.307} C_VEL
LIN {X 0,Y 592.022,Z 1195.103,A -85,B 0,C 180,E1 26900.963,E2 26900.963} C_VEL
LIN {X 0,Y 592.224,Z 1188.471,A -85,B 0,C 180,E1 26898.31,E2 26898.31} C_VEL
LIN {X 0,Y 592.556,Z 1180.571,A -85,B 0,C 180,E1 26895.838,E2 26895.838} C_VEL
LIN {X 0,Y 593.028,Z 1172.305,A -85,B 0,C 180,E1 26893.646,E2 26893.646} C_VEL
LIN {X 0,Y 593.709,Z 1162.694,A -85,B 0,C 180,E1 26891.44,E2 26891.44} C_VEL
LIN {X 0,Y 594.841,Z 1149.446,A -85,B 0,C 180,E1 26888.815,E2 26888.815} C_VEL
LIN {X 0,Y 596.107,Z 1136.315,A -85,B 0,C 180,E1 26886.567,E2 26886.567} C_VEL
LIN {X 0,Y 597.54,Z 1122.985,A -85,B 0,C 180,E1 26884.53,E2 26884.53} C_VEL
LIN {X 0,Y 599.573,Z 1106.413,A -85,B 0,C 180,E1 26882.273,E2 26882.273} C_VEL
LIN {X 0,Y 601.819,Z 1088.229,A -85,B 0,C 180,E1 26880.105,E2 26880.105} C_VEL
LIN {X 0,Y 603.941,Z 1072.291,A -85,B 0,C 180,E1 26878.4,E2 26878.4} C_VEL
LIN {X 0,Y 606.351,Z 1054.613,A -85,B 0,C 180,E1 26876.694,E2 26876.694} C_VEL
LIN {X 0,Y 609.496,Z 1031.566,A -85,B 0,C 180,E1 26874.729,E2 26874.729} C_VEL
LIN {X 0,Y 612.158,Z 1011.517,A -85,B 0,C 180,E1 26873.229,E2 26873.229} C_VEL
LIN {X 0,Y 614.692,Z 992.1,A -85,B 0,C 180,E1 26871.934,E2 26871.934} C_VEL
LIN {X 0,Y 617.675,Z 968.572,A -85,B 0,C 180,E1 26870.549,E2 26870.549} C_VEL
LIN {X 0,Y 620.469,Z 943.985,A -85,B 0,C 180,E1 26869.32,E2 26869.32} C_VEL
LIN {X 0,Y 622.709,Z 922.583,A -85,B 0,C 180,E1 26868.399,E2 26868.399} C_VEL
LIN {X 0,Y 624.662,Z 901.901,A -85,B 0,C 180,E1 26867.634,E2 26867.634} C_VEL
LIN {X 0,Y 626.528,Z 879.601,A -85,B 0,C 180,E1 26866.939,E2 26866.939} C_VEL
LIN {X 0,Y 628.497,Z 850.958,A -85,B 0,C 180,E1 26866.238,E2 26866.238} C_VEL
LIN {X 0,Y 629.693,Z 826.933,A -85,B 0,C 180,E1 26865.806,E2 26865.806} C_VEL
LIN {X 0,Y 633.809,Z 659.418,A -85,B 0,C 180,E1 26863.5,E2 26863.5} C_VEL
LIN {X 0,Y 639.319,Z 442.593,A -85,B 0,C 180,E1 26860.471,E2 26860.471} C_VEL
LIN {X 0,Y 640.077,Z 408.842,A -85,B 0,C 180,E1 26859.976,E2 26859.976} C_VEL
LIN {X 0,Y 626.243,Z 387.86,A -85,B 0,C 180,E1 26858.018,E2 26858.018} C_VEL
LIN {X 0,Y 616.601,Z 374.211,A -85,B 0,C 180,E1 26856.522,E2 26856.522} C_VEL
LIN {X 0,Y 606.89,Z 361.141,A -85,B 0,C 180,E1 26854.898,E2 26854.898} C_VEL
LIN {X 0,Y 603.21,Z 356.262,A -85,B 0,C 180,E1 26854.247,E2 26854.247} C_VEL
LIN {X 0,Y 599.006,Z 351.021,A -85,B 0,C 180,E1 26853.483,E2 26853.483} C_VEL
LIN {X 0,Y 597.117,Z 348.726,A -85,B 0,C 180,E1 26853.086,E2 26853.086} C_VEL
LIN {X 0,Y 595.49,Z 345.003,A -85,B 0,C 180,E1 26852.375,E2 26852.375} C_VEL
LIN {X 0,Y 593.406,Z 341.594,A -85,B 0,C 180,E1 26851.604,E2 26851.604} C_VEL
LIN {X 0,Y 593.124,Z 340.309,A -85,B 0,C 180,E1 26851.337,E2 26851.337} C_VEL
LIN {X 0,Y 593.178,Z 340.321,A -85,B 0,C 180,E1 26848.372,E2 26848.372} C_VEL
LIN {X 0,Y 593.131,Z 340.345,A -85,B 0,C 180,E1 26845.145,E2 26845.145} C_VEL
LIN {X 0,Y 593.198,Z 340.299,A -85,B 0,C 180,E1 26842.022,E2 26842.022} C_VEL
LIN {X 0,Y 593.13,Z 340.331,A -85,B 0,C 180,E1 26838.885,E2 26838.885} C_VEL
LIN {X 0,Y 593.201,Z 340.325,A -85,B 0,C 180,E1 26835.746,E2 26835.746} C_VEL
LIN {X 0,Y 593.128,Z 340.307,A -85,B 0,C 180,E1 26832.659,E2 26832.659} C_VEL
LIN {X 0,Y 593.199,Z 340.341,A -85,B 0,C 180,E1 26829.508,E2 26829.508} C_VEL
LIN {X 0,Y 593.128,Z 340.304,A -85,B 0,C 180,E1 26826.485,E2 26826.485} C_VEL
LIN {X 0,Y 593.197,Z 340.335,A -85,B 0,C 180,E1 26823.382,E2 26823.382} C_VEL
LIN {X 0,Y 593.131,Z 340.315,A -85,B 0,C 180,E1 26820.29,E2 26820.29} C_VEL
LIN {X 0,Y 593.196,Z 340.316,A -85,B 0,C 180,E1 26817.198,E2 26817.198} C_VEL
LIN {X 0,Y 593.134,Z 340.333,A -85,B 0,C 180,E1 26814.098,E2 26814.098} C_VEL
LIN {X 0,Y 593.196,Z 340.301,A -85,B 0,C 180,E1 26811.013,E2 26811.013} C_VEL
LIN {X 0,Y 593.139,Z 340.346,A -85,B 0,C 180,E1 26807.835,E2 26807.835} C_VEL
LIN {X 0,Y 593.191,Z 340.303,A -85,B 0,C 180,E1 26804.654,E2 26804.654} C_VEL
LIN {X 0,Y 593.139,Z 340.319,A -85,B 0,C 180,E1 26801.625,E2 26801.625} C_VEL
LIN {X 0,Y 593.197,Z 340.343,A -85,B 0,C 180,E1 26798.441,E2 26798.441} C_VEL
LIN {X 0,Y 593.14,Z 340.316,A -85,B 0,C 180,E1 26795.393,E2 26795.393} C_VEL
LIN {X 0,Y 593.222,Z 340.514,A -85,B 0,C 180,E1 26794.694,E2 26794.694} C_VEL
LIN {X 0,Y 594.023,Z 343.028,A -85,B 0,C 180,E1 26794.301,E2 26794.301} C_VEL
LIN {X 0,Y 596.209,Z 345.689,A -85,B 0,C 180,E1 26793.881,E2 26793.881} C_VEL
LIN {X 0,Y 597.602,Z 347.034,A -85,B 0,C 180,E1 26793.626,E2 26793.626} C_VEL
LIN {X 0,Y 601.519,Z 351.8,A -85,B 0,C 180,E1 26792.905,E2 26792.905} C_VEL
LIN {X 0,Y 610.925,Z 363.841,A -85,B 0,C 180,E1 26791.264,E2 26791.264} C_VEL
LIN {X 0,Y 621.168,Z 377.536,A -85,B 0,C 180,E1 26789.612,E2 26789.612} C_VEL
LIN {X 0,Y 631.988,Z 393.47,A -85,B 0,C 180,E1 26787.993,E2 26787.993} C_VEL
LIN {X 0,Y 640.1,Z 405.644,A -85,B 0,C 180,E1 26786.878,E2 26786.878} C_VEL
LIN {X 0,Y 634.931,Z 606.012,A -85,B 0,C 180,E1 26784.059,E2 26784.059} C_VEL
LIN {X 0,Y 634.057,Z 641.365,A -85,B 0,C 180,E1 26783.569,E2 26783.569} C_VEL
LIN {X 0,Y 633.18,Z 649.067,A -85,B 0,C 180,E1 26783.529,E2 26783.529} C_VEL
LIN {X 0,Y 628.365,Z 669.715,A -85,B 0,C 180,E1 26783.656,E2 26783.656} C_VEL
LIN {X 0,Y 627.664,Z 676.324,A -85,B 0,C 180,E1 26783.615,E2 26783.615} C_VEL
LIN {X 0,Y 623.92,Z 818.9,A -85,B 0,C 180,E1 26781.636,E2 26781.636} C_VEL
LIN {X 0,Y 622.304,Z 847.371,A -85,B 0,C 180,E1 26781.091,E2 26781.091} C_VEL
LIN {X 0,Y 620.551,Z 870.729,A -85,B 0,C 180,E1 26780.494,E2 26780.494} C_VEL
LIN {X 0,Y 618.609,Z 893.023,A -85,B 0,C 180,E1 26779.791,E2 26779.791} C_VEL
LIN {X 0,Y 615.827,Z 920.386,A -85,B 0,C 180,E1 26778.74,E2 26778.74} C_VEL
LIN {X 0,Y 613.31,Z 942.121,A -85,B 0,C 180,E1 26777.743,E2 26777.743} C_VEL
LIN {X 0,Y 610.693,Z 963.239,A -85,B 0,C 180,E1 26776.63,E2 26776.63} C_VEL
LIN {X 0,Y 607.563,Z 987.257,A -85,B 0,C 180,E1 26775.177,E2 26775.177} C_VEL
LIN {X 0,Y 604.419,Z 1009.488,A -85,B 0,C 180,E1 26773.616,E2 26773.616} C_VEL
LIN {X 0,Y 601.592,Z 1029.276,A -85,B 0,C 180,E1 26772.051,E2 26772.051} C_VEL
LIN {X 0,Y 598.346,Z 1051.66,A -85,B 0,C 180,E1 26770.042,E2 26770.042} C_VEL
LIN {X 0,Y 595.703,Z 1070.197,A -85,B 0,C 180,E1 26768.146,E2 26768.146} C_VEL
LIN {X 0,Y 593.173,Z 1088.634,A -85,B 0,C 180,E1 26766.035,E2 26766.035} C_VEL
LIN {X 0,Y 590.827,Z 1106.389,A -85,B 0,C 180,E1 26763.716,E2 26763.716} C_VEL
LIN {X 0,Y 588.9,Z 1122.448,A -85,B 0,C 180,E1 26761.345,E2 26761.345} C_VEL
LIN {X 0,Y 587.274,Z 1137.417,A -85,B 0,C 180,E1 26758.804,E2 26758.804} C_VEL
LIN {X 0,Y 586.037,Z 1150.624,A -85,B 0,C 180,E1 26756.224,E2 26756.224} C_VEL
LIN {X 0,Y 585.117,Z 1162.643,A -85,B 0,C 180,E1 26753.463,E2 26753.463} C_VEL
LIN {X 0,Y 584.568,Z 1171.484,A -85,B 0,C 180,E1 26751.05,E2 26751.05} C_VEL
LIN {X 0,Y 584.218,Z 1179.248,A -85,B 0,C 180,E1 26748.526,E2 26748.526} C_VEL
LIN {X 0,Y 584.024,Z 1185.567,A -85,B 0,C 180,E1 26745.898,E2 26745.898} C_VEL
LIN {X 0,Y 583.947,Z 1189.817,A -85,B 0,C 180,E1 26743.567,E2 26743.567} C_VEL
LIN {X 0,Y 583.915,Z 1193.008,A -85,B 0,C 180,E1 26741.057,E2 26741.057} C_VEL
LIN {X 0,Y 583.912,Z 1194.664,A -85,B 0,C 180,E1 26738.468,E2 26738.468} C_VEL
LIN {X 0,Y 583.913,Z 1194.835,A -85,B 0,C 180,E1 26736.193,E2 26736.193} C_VEL
LIN {X 0,Y 583.911,Z 1193.936,A -85,B 0,C 180,E1 26734.026,E2 26734.026} C_VEL
LIN {X 0,Y 583.921,Z 1191.585,A -85,B 0,C 180,E1 26731.57,E2 26731.57} C_VEL
LIN {X 0,Y 583.99,Z 1187.401,A -85,B 0,C 180,E1 26728.921,E2 26728.921} C_VEL
LIN {X 0,Y 584.109,Z 1182.254,A -85,B 0,C 180,E1 26726.565,E2 26726.565} C_VEL
LIN {X 0,Y 584.353,Z 1175.802,A -85,B 0,C 180,E1 26724.206,E2 26724.206} C_VEL
LIN {X 0,Y 584.822,Z 1166.906,A -85,B 0,C 180,E1 26721.545,E2 26721.545} C_VEL
LIN {X 0,Y 585.598,Z 1156.03,A -85,B 0,C 180,E1 26718.876,E2 26718.876} C_VEL
LIN {X 0,Y 586.591,Z 1144.271,A -85,B 0,C 180,E1 26716.395,E2 26716.395} C_VEL
LIN {X 0,Y 587.968,Z 1130.593,A -85,B 0,C 180,E1 26713.908,E2 26713.908} C_VEL
LIN {X 0,Y 589.68,Z 1115.602,A -85,B 0,C 180,E1 26711.514,E2 26711.514} C_VEL
LIN {X 0,Y 591.958,Z 1097.647,A -85,B 0,C 180,E1 26709.018,E2 26709.018} C_VEL
LIN {X 0,Y 594.235,Z 1080.548,A -85,B 0,C 180,E1 26706.918,E2 26706.918} C_VEL
LIN {X 0,Y 597.141,Z 1060.26,A -85,B 0,C 180,E1 26704.718,E2 26704.718} C_VEL
LIN {X 0,Y 599.89,Z 1041.013,A -85,B 0,C 180,E1 26702.882,E2 26702.882} C_VEL
LIN {X 0,Y 602.928,Z 1019.982,A -85,B 0,C 180,E1 26701.092,E2 26701.092} C_VEL
LIN {X 0,Y 606.122,Z 997.315,A -85,B 0,C 180,E1 26699.415,E2 26699.415} C_VEL
LIN {X 0,Y 608.917,Z 976.834,A -85,B 0,C 180,E1 26698.08,E2 26698.08} C_VEL
LIN {X 0,Y 611.943,Z 953.865,A -85,B 0,C 180,E1 26696.764,E2 26696.764} C_VEL
LIN {X 0,Y 614.911,Z 928.727,A -85,B 0,C 180,E1 26695.538,E2 26695.538} C_VEL
LIN {X 0,Y 617.123,Z 907.811,A -85,B 0,C 180,E1 26694.661,E2 26694.661} C_VEL
LIN {X 0,Y 619.243,Z 886.172,A -85,B 0,C 180,E1 26693.89,E2 26693.89} C_VEL
LIN {X 0,Y 621.506,Z 859.011,A -85,B 0,C 180,E1 26693.096,E2 26693.096} C_VEL
LIN {X 0,Y 623.108,Z 834.017,A -85,B 0,C 180,E1 26692.54,E2 26692.54} C_VEL
LIN {X 0,Y 624.27,Z 809.787,A -85,B 0,C 180,E1 26692.137,E2 26692.137} C_VEL
LIN {X 0,Y 629.907,Z 590.118,A -85,B 0,C 180,E1 26689.092,E2 26689.092} C_VEL
LIN {X 0,Y 634.813,Z 409.54,A -85,B 0,C 180,E1 26686.53,E2 26686.53} C_VEL
LIN {X 0,Y 621.662,Z 390.49,A -85,B 0,C 180,E1 26684.723,E2 26684.723} C_VEL
LIN {X 0,Y 607.819,Z 371.76,A -85,B 0,C 180,E1 26682.733,E2 26682.733} C_VEL
LIN {X 0,Y 596.977,Z 357.407,A -85,B 0,C 180,E1 26681.071,E2 26681.071} C_VEL
LIN {X 0,Y 593.167,Z 352.644,A -85,B 0,C 180,E1 26680.466,E2 26680.466} C_VEL
LIN {X 0,Y 590.378,Z 349.162,A -85,B 0,C 180,E1 26680.012,E2 26680.012} C_VEL
LIN {X 0,Y 589.051,Z 347.201,A -85,B 0,C 180,E1 26679.788,E2 26679.788} C_VEL
LIN {X 0,Y 586.307,Z 344.489,A -85,B 0,C 180,E1 26679.345,E2 26679.345} C_VEL
LIN {X 0,Y 585.345,Z 342.209,A -85,B 0,C 180,E1 26679.15,E2 26679.15} C_VEL
LIN {X 0,Y 585.172,Z 341.334,A -85,B 0,C 180,E1 26678.974,E2 26678.974} C_VEL
LIN {X 0,Y 585.183,Z 341.339,A -85,B 0,C 180,E1 26676.082,E2 26676.082} C_VEL
LIN {X 0,Y 585.173,Z 341.336,A -85,B 0,C 180,E1 26672.791,E2 26672.791} C_VEL
LIN {X 0,Y 585.185,Z 341.328,A -85,B 0,C 180,E1 26669.93,E2 26669.93} C_VEL
LIN {X 0,Y 585.17,Z 341.302,A -85,B 0,C 180,E1 26666.595,E2 26666.595} C_VEL
LIN {X 0,Y 585.192,Z 341.319,A -85,B 0,C 180,E1 26663.674,E2 26663.674} C_VEL
LIN {X 0,Y 585.169,Z 341.3,A -85,B 0,C 180,E1 26660.401,E2 26660.401} C_VEL
LIN {X 0,Y 585.197,Z 341.331,A -85,B 0,C 180,E1 26657.501,E2 26657.501} C_VEL
LIN {X 0,Y 585.174,Z 341.333,A -85,B 0,C 180,E1 26654.244,E2 26654.244} C_VEL
LIN {X 0,Y 585.196,Z 341.338,A -85,B 0,C 180,E1 26651.332,E2 26651.332} C_VEL
LIN {X 0,Y 585.176,Z 341.337,A -85,B 0,C 180,E1 26648.054,E2 26648.054} C_VEL
LIN {X 0,Y 585.187,Z 341.328,A -85,B 0,C 180,E1 26645.294,E2 26645.294} C_VEL
LIN {X 0,Y 585.18,Z 341.33,A -85,B 0,C 180,E1 26641.958,E2 26641.958} C_VEL
LIN {X 0,Y 585.182,Z 341.325,A -85,B 0,C 180,E1 26639.217,E2 26639.217} C_VEL
LIN {X 0,Y 585.186,Z 341.322,A -85,B 0,C 180,E1 26635.885,E2 26635.885} C_VEL
LIN {X 0,Y 585.186,Z 341.336,A -85,B 0,C 180,E1 26633.032,E2 26633.032} C_VEL
LIN {X 0,Y 585.186,Z 341.332,A -85,B 0,C 180,E1 26629.665,E2 26629.665} C_VEL
LIN {X 0,Y 585.191,Z 341.279,A -85,B 0,C 180,E1 26626.764,E2 26626.764} C_VEL
LIN {X 0,Y 585.185,Z 341.335,A -85,B 0,C 180,E1 26623.442,E2 26623.442} C_VEL
LIN {X 0,Y 585.198,Z 341.282,A -85,B 0,C 180,E1 26620.538,E2 26620.538} C_VEL
LIN {X 0,Y 585.186,Z 341.332,A -85,B 0,C 180,E1 26617.284,E2 26617.284} C_VEL
LIN {X 0,Y 585.199,Z 341.289,A -85,B 0,C 180,E1 26614.387,E2 26614.387} C_VEL
LIN {X 0,Y 585.186,Z 341.328,A -85,B 0,C 180,E1 26611.082,E2 26611.082} C_VEL
LIN {X 0,Y 585.204,Z 341.501,A -85,B 0,C 180,E1 26608.68,E2 26608.68} C_VEL
LIN {X 0,Y 586.585,Z 344.905,A -85,B 0,C 180,E1 26608.101,E2 26608.101} C_VEL
LIN {X 0,Y 587.628,Z 346.117,A -85,B 0,C 180,E1 26607.819,E2 26607.819} C_VEL
LIN {X 0,Y 589.284,Z 349.847,A -85,B 0,C 180,E1 26607.229,E2 26607.229} C_VEL
LIN {X 0,Y 594.287,Z 356.091,A -85,B 0,C 180,E1 26606.418,E2 26606.418} C_VEL
LIN {X 0,Y 610.347,Z 377.92,A -85,B 0,C 180,E1 26603.947,E2 26603.947} C_VEL
LIN {X 0,Y 624.525,Z 397.556,A -85,B 0,C 180,E1 26601.931,E2 26601.931} C_VEL
LIN {X 0,Y 634.933,Z 413.04,A -85,B 0,C 180,E1 26600.507,E2 26600.507} C_VEL
LIN {X 0,Y 629.411,Z 616.656,A -85,B 0,C 180,E1 26597.626,E2 26597.626} C_VEL
LIN {X 0,Y 624.012,Z 825.273,A -85,B 0,C 180,E1 26594.731,E2 26594.731} C_VEL
LIN {X 0,Y 622.882,Z 847.356,A -85,B 0,C 180,E1 26594.344,E2 26594.344} C_VEL
LIN {X 0,Y 621.244,Z 872.232,A -85,B 0,C 180,E1 26593.771,E2 26593.771} C_VEL
LIN {X 0,Y 618.938,Z 899.277,A -85,B 0,C 180,E1 26592.961,E2 26592.961} C_VEL
LIN {X 0,Y 616.84,Z 920.635,A -85,B 0,C 180,E1 26592.181,E2 26592.181} C_VEL
LIN {X 0,Y 614.683,Z 940.588,A -85,B 0,C 180,E1 26591.331,E2 26591.331} C_VEL
LIN {X 0,Y 612.542,Z 958.685,A -85,B 0,C 180,E1 26590.454,E2 26590.454} C_VEL
LIN {X 0,Y 610.137,Z 977.635,A -85,B 0,C 180,E1 26589.421,E2 26589.421} C_VEL
LIN {X 0,Y 607.445,Z 997.869,A -85,B 0,C 180,E1 26588.176,E2 26588.176} C_VEL
LIN {X 0,Y 603.998,Z 1022.552,A -85,B 0,C 180,E1 26586.433,E2 26586.433} C_VEL
LIN {X 0,Y 601.133,Z 1042.225,A -85,B 0,C 180,E1 26584.844,E2 26584.844} C_VEL
LIN {X 0,Y 598.62,Z 1059.608,A -85,B 0,C 180,E1 26583.277,E2 26583.277} C_VEL
LIN {X 0,Y 595.843,Z 1079.333,A -85,B 0,C 180,E1 26581.295,E2 26581.295} C_VEL
LIN {X 0,Y 593.241,Z 1097.991,A -85,B 0,C 180,E1 26579.149,E2 26579.149} C_VEL
LIN {X 0,Y 591.276,Z 1112.615,A -85,B 0,C 180,E1 26577.275,E2 26577.275} C_VEL
LIN {X 0,Y 589.498,Z 1127.186,A -85,B 0,C 180,E1 26575.196,E2 26575.196} C_VEL
LIN {X 0,Y 587.644,Z 1143.706,A -85,B 0,C 180,E1 26572.509,E2 26572.509} C_VEL
LIN {X 0,Y 586.477,Z 1155.376,A -85,B 0,C 180,E1 26570.33,E2 26570.33} C_VEL
LIN {X 0,Y 585.631,Z 1165.448,A -85,B 0,C 180,E1 26568.206,E2 26568.206} C_VEL
LIN {X 0,Y 584.857,Z 1176.307,A -85,B 0,C 180,E1 26565.569,E2 26565.569} C_VEL
LIN {X 0,Y 584.389,Z 1185.177,A -85,B 0,C 180,E1 26562.952,E2 26562.952} C_VEL
LIN {X 0,Y 584.128,Z 1191.603,A -85,B 0,C 180,E1 26560.653,E2 26560.653} C_VEL
LIN {X 0,Y 583.992,Z 1197.151,A -85,B 0,C 180,E1 26558.17,E2 26558.17} C_VEL
LIN {X 0,Y 583.93,Z 1201.428,A -85,B 0,C 180,E1 26555.502,E2 26555.502} C_VEL
LIN {X 0,Y 583.917,Z 1203.854,A -85,B 0,C 180,E1 26553.043,E2 26553.043} C_VEL
LIN {X 0,Y 583.905,Z 1204.804,A -85,B 0,C 180,E1 26550.883,E2 26550.883} C_VEL
LIN {X 0,Y 583.915,Z 1204.736,A -85,B 0,C 180,E1 26548.823,E2 26548.823} C_VEL
LIN {X 0,Y 583.913,Z 1203.51,A -85,B 0,C 180,E1 26546.466,E2 26546.466} C_VEL
LIN {X 0,Y 583.943,Z 1200.337,A -85,B 0,C 180,E1 26543.709,E2 26543.709} C_VEL
LIN {X 0,Y 584.019,Z 1195.926,A -85,B 0,C 180,E1 26541.236,E2 26541.236} C_VEL
LIN {X 0,Y 584.152,Z 1190.586,A -85,B 0,C 180,E1 26538.948,E2 26538.948} C_VEL
LIN {X 0,Y 584.519,Z 1182.685,A -85,B 0,C 180,E1 26536.245,E2 26536.245} C_VEL
LIN {X 0,Y 585.07,Z 1173.113,A -85,B 0,C 180,E1 26533.622,E2 26533.622} C_VEL
LIN {X 0,Y 585.743,Z 1164.074,A -85,B 0,C 180,E1 26531.488,E2 26531.488} C_VEL
LIN {X 0,Y 586.693,Z 1153.206,A -85,B 0,C 180,E1 26529.239,E2 26529.239} C_VEL
LIN {X 0,Y 588.226,Z 1138.277,A -85,B 0,C 180,E1 26526.562,E2 26526.562} C_VEL
LIN {X 0,Y 589.783,Z 1124.56,A -85,B 0,C 180,E1 26524.413,E2 26524.413} C_VEL
LIN {X 0,Y 591.601,Z 1110.302,A -85,B 0,C 180,E1 26522.414,E2 26522.414} C_VEL
LIN {X 0,Y 594.11,Z 1091.609,A -85,B 0,C 180,E1 26520.083,E2 26520.083} C_VEL
LIN {X 0,Y 596.592,Z 1073.81,A -85,B 0,C 180,E1 26518.135,E2 26518.135} C_VEL
LIN {X 0,Y 598.947,Z 1057.387,A -85,B 0,C 180,E1 26516.515,E2 26516.515} C_VEL
LIN {X 0,Y 601.698,Z 1038.571,A -85,B 0,C 180,E1 26514.845,E2 26514.845} C_VEL
LIN {X 0,Y 605.028,Z 1015.188,A -85,B 0,C 180,E1 26513.02,E2 26513.02} C_VEL
LIN {X 0,Y 607.749,Z 995.427,A -85,B 0,C 180,E1 26511.667,E2 26511.667} C_VEL
LIN {X 0,Y 610.362,Z 975.836,A -85,B 0,C 180,E1 26510.475,E2 26510.475} C_VEL
LIN {X 0,Y 612.906,Z 955.676,A -85,B 0,C 180,E1 26509.39,E2 26509.39} C_VEL
LIN {X 0,Y 615.754,Z 931.539,A -85,B 0,C 180,E1 26508.26,E2 26508.26} C_VEL
LIN {X 0,Y 618.271,Z 906.288,A -85,B 0,C 180,E1 26507.281,E2 26507.281} C_VEL
LIN {X 0,Y 620.181,Z 884.888,A -85,B 0,C 180,E1 26506.587,E2 26506.587} C_VEL
LIN {X 0,Y 621.808,Z 863.786,A -85,B 0,C 180,E1 26506.021,E2 26506.021} C_VEL
LIN {X 0,Y 623.158,Z 842.379,A -85,B 0,C 180,E1 26505.558,E2 26505.558} C_VEL
LIN {X 0,Y 624.412,Z 815.237,A -85,B 0,C 180,E1 26505.117,E2 26505.117} C_VEL
LIN {X 0,Y 630.017,Z 593.12,A -85,B 0,C 180,E1 26502.046,E2 26502.046} C_VEL
LIN {X 0,Y 634.904,Z 412.832,A -85,B 0,C 180,E1 26499.484,E2 26499.484} C_VEL
LIN {X 0,Y 620.718,Z 391.277,A -85,B 0,C 180,E1 26497.394,E2 26497.394} C_VEL
LIN {X 0,Y 610.926,Z 377.259,A -85,B 0,C 180,E1 26495.811,E2 26495.811} C_VEL
LIN {X 0,Y 603.297,Z 367.26,A -85,B 0,C 180,E1 26494.5,E2 26494.5} C_VEL
LIN {X 0,Y 599.085,Z 361.72,A -85,B 0,C 180,E1 26493.736,E2 26493.736} C_VEL
LIN {X 0,Y 594.505,Z 355.967,A -85,B 0,C 180,E1 26492.877,E2 26492.877} C_VEL
LIN {X 0,Y 590.16,Z 350.575,A -85,B 0,C 180,E1 26492.026,E2 26492.026} C_VEL
LIN {X 0,Y 588.606,Z 348.531,A -85,B 0,C 180,E1 26491.662,E2 26491.662} C_VEL
LIN {X 0,Y 587.532,Z 346.028,A -85,B 0,C 180,E1 26491.156,E2 26491.156} C_VEL
LIN {X 0,Y 585.686,Z 343.128,A -85,B 0,C 180,E1 26490.445,E2 26490.445} C_VEL
LIN {X 0,Y 585.262,Z 341.301,A -85,B 0,C 180,E1 26490.111,E2 26490.111} C_VEL
LIN {X 0,Y 585.185,Z 341.295,A -85,B 0,C 180,E1 26487.033,E2 26487.033} C_VEL
LIN {X 0,Y 585.256,Z 341.311,A -85,B 0,C 180,E1 26483.885,E2 26483.885} C_VEL
LIN {X 0,Y 585.191,Z 341.32,A -85,B 0,C 180,E1 26480.818,E2 26480.818} C_VEL
LIN {X 0,Y 585.25,Z 341.287,A -85,B 0,C 180,E1 26477.705,E2 26477.705} C_VEL
LIN {X 0,Y 585.193,Z 341.336,A -85,B 0,C 180,E1 26474.648,E2 26474.648} C_VEL
LIN {X 0,Y 585.253,Z 341.287,A -85,B 0,C 180,E1 26471.531,E2 26471.531} C_VEL
LIN {X 0,Y 585.194,Z 341.323,A -85,B 0,C 180,E1 26468.45,E2 26468.45} C_VEL
LIN {X 0,Y 585.25,Z 341.305,A -85,B 0,C 180,E1 26465.294,E2 26465.294} C_VEL
LIN {X 0,Y 585.192,Z 341.303,A -85,B 0,C 180,E1 26462.252,E2 26462.252} C_VEL
LIN {X 0,Y 585.248,Z 341.325,A -85,B 0,C 180,E1 26459.021,E2 26459.021} C_VEL
LIN {X 0,Y 585.195,Z 341.29,A -85,B 0,C 180,E1 26455.983,E2 26455.983} C_VEL
LIN {X 0,Y 585.238,Z 341.329,A -85,B 0,C 180,E1 26452.737,E2 26452.737} C_VEL
LIN {X 0,Y 585.206,Z 341.297,A -85,B 0,C 180,E1 26449.665,E2 26449.665} C_VEL
LIN {X 0,Y 585.215,Z 341.3,A -85,B 0,C 180,E1 26446.362,E2 26446.362} C_VEL
LIN {X 0,Y 585.214,Z 341.33,A -85,B 0,C 180,E1 26443.421,E2 26443.421} C_VEL
LIN {X 0,Y 585.212,Z 341.296,A -85,B 0,C 180,E1 26440.122,E2 26440.122} C_VEL
LIN {X 0,Y 585.218,Z 341.304,A -85,B 0,C 180,E1 26437.179,E2 26437.179} C_VEL
LIN {X 0,Y 585.218,Z 341.337,A -85,B 0,C 180,E1 26436.006,E2 26436.006} C_VEL
LIN {X 0,Y 585.729,Z 343.33,A -85,B 0,C 180,E1 26435.719,E2 26435.719} C_VEL
LIN {X 0,Y 587.574,Z 346.061,A -85,B 0,C 180,E1 26435.325,E2 26435.325} C_VEL
LIN {X 0,Y 590.143,Z 348.095,A -85,B 0,C 180,E1 26434.832,E2 26434.832} C_VEL
LIN {X 0,Y 593.171,Z 352.406,A -85,B 0,C 180,E1 26434.221,E2 26434.221} C_VEL
LIN {X 0,Y 595.231,Z 354.512,A -85,B 0,C 180,E1 26433.835,E2 26433.835} C_VEL
LIN {X 0,Y 603.781,Z 365.274,A -85,B 0,C 180,E1 26432.267,E2 26432.267} C_VEL
LIN {X 0,Y 608.562,Z 371.56,A -85,B 0,C 180,E1 26431.437,E2 26431.437} C_VEL
LIN {X 0,Y 617.849,Z 384.053,A -85,B 0,C 180,E1 26429.915,E2 26429.915} C_VEL
LIN {X 0,Y 628.798,Z 400.372,A -85,B 0,C 180,E1 26428.241,E2 26428.241} C_VEL
LIN {X 0,Y 634.867,Z 409.751,A -85,B 0,C 180,E1 26427.375,E2 26427.375} C_VEL
LIN {X 0,Y 629.231,Z 615.982,A -85,B 0,C 180,E1 26424.455,E2 26424.455} C_VEL
LIN {X 0,Y 627.664,Z 676.324,A -85,B 0,C 180,E1 26423.615,E2 26423.615} C_VEL
LIN {X 0,Y 626.768,Z 684.027,A -85,B 0,C 180,E1 26423.576,E2 26423.576} C_VEL
LIN {X 0,Y 621.94,Z 704.665,A -85,B 0,C 180,E1 26423.707,E2 26423.707} C_VEL
LIN {X 0,Y 621.23,Z 711.273,A -85,B 0,C 180,E1 26423.667,E2 26423.667} C_VEL
LIN {X 0,Y 618.221,Z 819.101,A -85,B 0,C 180,E1 26422.155,E2 26422.155} C_VEL
LIN {X 0,Y 616.555,Z 847.348,A -85,B 0,C 180,E1 26421.614,E2 26421.614} C_VEL
LIN {X 0,Y 614.656,Z 871.567,A -85,B 0,C 180,E1 26420.99,E2 26420.99} C_VEL
LIN {X 0,Y 612.417,Z 896.009,A -85,B 0,C 180,E1 26420.207,E2 26420.207} C_VEL
LIN {X 0,Y 609.611,Z 921.732,A -85,B 0,C 180,E1 26419.194,E2 26419.194} C_VEL
LIN {X 0,Y 606.962,Z 943.365,A -85,B 0,C 180,E1 26418.187,E2 26418.187} C_VEL
LIN {X 0,Y 604.236,Z 964.237,A -85,B 0,C 180,E1 26417.073,E2 26417.073} C_VEL
LIN {X 0,Y 600.722,Z 989.498,A -85,B 0,C 180,E1 26415.513,E2 26415.513} C_VEL
LIN {X 0,Y 597.756,Z 1009.468,A -85,B 0,C 180,E1 26414.094,E2 26414.094} C_VEL
LIN {X 0,Y 594.924,Z 1028.287,A -85,B 0,C 180,E1 26412.595,E2 26412.595} C_VEL
LIN {X 0,Y 591.584,Z 1050.168,A -85,B 0,C 180,E1 26410.633,E2 26410.633} C_VEL
LIN {X 0,Y 588.669,Z 1069.137,A -85,B 0,C 180,E1 26408.686,E2 26408.686} C_VEL
LIN {X 0,Y 586.028,Z 1087.407,A -85,B 0,C 180,E1 26406.584,E2 26406.584} C_VEL
LIN {X 0,Y 583.438,Z 1105.584,A -85,B 0,C 180,E1 26404.201,E2 26404.201} C_VEL
LIN {X 0,Y 581.42,Z 1121.285,A -85,B 0,C 180,E1 26401.866,E2 26401.866} C_VEL
LIN {X 0,Y 579.579,Z 1136.965,A -85,B 0,C 180,E1 26399.196,E2 26399.196} C_VEL
LIN {X 0,Y 578.292,Z 1149.573,A -85,B 0,C 180,E1 26396.714,E2 26396.714} C_VEL
LIN {X 0,Y 577.318,Z 1160.995,A -85,B 0,C 180,E1 26394.112,E2 26394.112} C_VEL
LIN {X 0,Y 576.695,Z 1170.418,A -85,B 0,C 180,E1 26391.565,E2 26391.565} C_VEL
LIN {X 0,Y 576.299,Z 1177.643,A -85,B 0,C 180,E1 26389.247,E2 26389.247} C_VEL
LIN {X 0,Y 576.08,Z 1184.282,A -85,B 0,C 180,E1 26386.641,E2 26386.641} C_VEL
LIN {X 0,Y 575.96,Z 1189.183,A -85,B 0,C 180,E1 26384.066,E2 26384.066} C_VEL
LIN {X 0,Y 575.917,Z 1192.368,A -85,B 0,C 180,E1 26381.705,E2 26381.705} C_VEL
LIN {X 0,Y 575.914,Z 1194.408,A -85,B 0,C 180,E1 26379.191,E2 26379.191} C_VEL
LIN {X 0,Y 575.908,Z 1194.901,A -85,B 0,C 180,E1 26376.48,E2 26376.48} C_VEL
LIN {X 0,Y 575.911,Z 1194.064,A -85,B 0,C 180,E1 26374.182,E2 26374.182} C_VEL
LIN {X 0,Y 575.923,Z 1191.91,A -85,B 0,C 180,E1 26371.791,E2 26371.791} C_VEL
LIN {X 0,Y 575.984,Z 1187.973,A -85,B 0,C 180,E1 26369.105,E2 26369.105} C_VEL
LIN {X 0,Y 576.118,Z 1182.491,A -85,B 0,C 180,E1 26366.518,E2 26366.518} C_VEL
LIN {X 0,Y 576.363,Z 1176.374,A -85,B 0,C 180,E1 26364.225,E2 26364.225} C_VEL
LIN {X 0,Y 576.792,Z 1168.657,A -85,B 0,C 180,E1 26361.828,E2 26361.828} C_VEL
LIN {X 0,Y 577.552,Z 1158.193,A -85,B 0,C 180,E1 26359.123,E2 26359.123} C_VEL
LIN {X 0,Y 578.554,Z 1146.754,A -85,B 0,C 180,E1 26356.61,E2 26356.61} C_VEL
LIN {X 0,Y 580.021,Z 1132.965,A -85,B 0,C 180,E1 26353.99,E2 26353.99} C_VEL
LIN {X 0,Y 581.782,Z 1118.209,A -85,B 0,C 180,E1 26351.565,E2 26351.565} C_VEL
LIN {X 0,Y 583.95,Z 1102.048,A -85,B 0,C 180,E1 26349.214,E2 26349.214} C_VEL
LIN {X 0,Y 586.358,Z 1084.81,A -85,B 0,C 180,E1 26347.015,E2 26347.015} C_VEL
LIN {X 0,Y 588.998,Z 1067.029,A -85,B 0,C 180,E1 26344.995,E2 26344.995} C_VEL
LIN {X 0,Y 592.321,Z 1045.366,A -85,B 0,C 180,E1 26342.826,E2 26342.826} C_VEL
LIN {X 0,Y 595.259,Z 1026.01,A -85,B 0,C 180,E1 26341.124,E2 26341.124} C_VEL
LIN {X 0,Y 598.34,Z 1005.628,A -85,B 0,C 180,E1 26339.525,E2 26339.525} C_VEL
LIN {X 0,Y 601.818,Z 981.619,A -85,B 0,C 180,E1 26337.883,E2 26337.883} C_VEL
LIN {X 0,Y 604.683,Z 960.843,A -85,B 0,C 180,E1 26336.647,E2 26336.647} C_VEL
LIN {X 0,Y 607.499,Z 939.209,A -85,B 0,C 180,E1 26335.516,E2 26335.516} C_VEL
LIN {X 0,Y 610.62,Z 912.849,A -85,B 0,C 180,E1 26334.343,E2 26334.343} C_VEL
LIN {X 0,Y 613.005,Z 889.792,A -85,B 0,C 180,E1 26333.492,E2 26333.492} C_VEL
LIN {X 0,Y 615.167,Z 865.811,A -85,B 0,C 180,E1 26332.758,E2 26332.758} C_VEL
LIN {X 0,Y 617.2,Z 837.459,A -85,B 0,C 180,E1 26332.085,E2 26332.085} C_VEL
LIN {X 0,Y 618.459,Z 813.276,A -85,B 0,C 180,E1 26331.665,E2 26331.665} C_VEL
LIN {X 0,Y 624.367,Z 596.498,A -85,B 0,C 180,E1 26328.635,E2 26328.635} C_VEL
LIN {X 0,Y 629.615,Z 413.436,A -85,B 0,C 180,E1 26326.026,E2 26326.026} C_VEL
LIN {X 0,Y 615.322,Z 393.021,A -85,B 0,C 180,E1 26324.035,E2 26324.035} C_VEL
LIN {X 0,Y 599.777,Z 372.102,A -85,B 0,C 180,E1 26321.728,E2 26321.728} C_VEL
LIN {X 0,Y 590.323,Z 359.699,A -85,B 0,C 180,E1 26320.223,E2 26320.223} C_VEL
LIN {X 0,Y 587.025,Z 355.616,A -85,B 0,C 180,E1 26319.681,E2 26319.681} C_VEL
LIN {X 0,Y 585.825,Z 354.02,A -85,B 0,C 180,E1 26319.479,E2 26319.479} C_VEL
LIN {X 0,Y 582.818,Z 350.624,A -85,B 0,C 180,E1 26318.976,E2 26318.976} C_VEL
LIN {X 0,Y 581.547,Z 348.472,A -85,B 0,C 180,E1 26318.745,E2 26318.745} C_VEL
LIN {X 0,Y 578.712,Z 346.062,A -85,B 0,C 180,E1 26318.273,E2 26318.273} C_VEL
LIN {X 0,Y 577.386,Z 343.087,A -85,B 0,C 180,E1 26318.009,E2 26318.009} C_VEL
LIN {X 0,Y 577.262,Z 342.328,A -85,B 0,C 180,E1 26317.945,E2 26317.945} C_VEL
LIN {X 0,Y 577.228,Z 342.319,A -85,B 0,C 180,E1 26314.744,E2 26314.744} C_VEL
LIN {X 0,Y 577.269,Z 342.314,A -85,B 0,C 180,E1 26311.741,E2 26311.741} C_VEL
LIN {X 0,Y 577.225,Z 342.279,A -85,B 0,C 180,E1 26308.561,E2 26308.561} C_VEL
LIN {X 0,Y 577.26,Z 342.314,A -85,B 0,C 180,E1 26305.66,E2 26305.66} C_VEL
LIN {X 0,Y 577.226,Z 342.275,A -85,B 0,C 180,E1 26302.401,E2 26302.401} C_VEL
LIN {X 0,Y 577.269,Z 342.309,A -85,B 0,C 180,E1 26299.425,E2 26299.425} C_VEL
LIN {X 0,Y 577.231,Z 342.318,A -85,B 0,C 180,E1 26296.194,E2 26296.194} C_VEL
LIN {X 0,Y 577.264,Z 342.311,A -85,B 0,C 180,E1 26293.319,E2 26293.319} C_VEL
LIN {X 0,Y 577.235,Z 342.312,A -85,B 0,C 180,E1 26290.076,E2 26290.076} C_VEL
LIN {X 0,Y 577.277,Z 342.316,A -85,B 0,C 180,E1 26287.064,E2 26287.064} C_VEL
LIN {X 0,Y 577.237,Z 342.324,A -85,B 0,C 180,E1 26283.874,E2 26283.874} C_VEL
LIN {X 0,Y 577.307,Z 342.322,A -85,B 0,C 180,E1 26280.695,E2 26280.695} C_VEL
LIN {X 0,Y 577.234,Z 342.326,A -85,B 0,C 180,E1 26277.518,E2 26277.518} C_VEL
LIN {X 0,Y 577.305,Z 342.316,A -85,B 0,C 180,E1 26274.334,E2 26274.334} C_VEL
LIN {X 0,Y 577.235,Z 342.32,A -85,B 0,C 180,E1 26271.332,E2 26271.332} C_VEL
LIN {X 0,Y 577.303,Z 342.273,A -85,B 0,C 180,E1 26268.207,E2 26268.207} C_VEL
LIN {X 0,Y 577.236,Z 342.307,A -85,B 0,C 180,E1 26265.135,E2 26265.135} C_VEL
LIN {X 0,Y 577.305,Z 342.278,A -85,B 0,C 180,E1 26262.043,E2 26262.043} C_VEL
LIN {X 0,Y 577.238,Z 342.308,A -85,B 0,C 180,E1 26258.988,E2 26258.988} C_VEL
LIN {X 0,Y 577.306,Z 342.268,A -85,B 0,C 180,E1 26255.873,E2 26255.873} C_VEL
LIN {X 0,Y 577.248,Z 342.327,A -85,B 0,C 180,E1 26252.694,E2 26252.694} C_VEL
LIN {X 0,Y 577.343,Z 342.481,A -85,B 0,C 180,E1 26249.736,E2 26249.736} C_VEL
LIN {X 0,Y 578.695,Z 345.994,A -85,B 0,C 180,E1 26249.125,E2 26249.125} C_VEL
LIN {X 0,Y 579.868,Z 347.906,A -85,B 0,C 180,E1 26248.733,E2 26248.733} C_VEL
LIN {X 0,Y 580.912,Z 349.986,A -85,B 0,C 180,E1 26248.42,E2 26248.42} C_VEL
LIN {X 0,Y 584.025,Z 353.849,A -85,B 0,C 180,E1 26247.886,E2 26247.886} C_VEL
LIN {X 0,Y 592.375,Z 364.775,A -85,B 0,C 180,E1 26246.499,E2 26246.499} C_VEL
LIN {X 0,Y 603.74,Z 380.096,A -85,B 0,C 180,E1 26244.719,E2 26244.719} C_VEL
LIN {X 0,Y 619.611,Z 401.978,A -85,B 0,C 180,E1 26242.411,E2 26242.411} C_VEL
LIN {X 0,Y 629.692,Z 417.118,A -85,B 0,C 180,E1 26241.01,E2 26241.01} C_VEL
LIN {X 0,Y 623.88,Z 621.412,A -85,B 0,C 180,E1 26238.103,E2 26238.103} C_VEL
LIN {X 0,Y 618.282,Z 826.059,A -85,B 0,C 180,E1 26235.241,E2 26235.241} C_VEL
LIN {X 0,Y 617.04,Z 848.986,A -85,B 0,C 180,E1 26234.832,E2 26234.832} C_VEL
LIN {X 0,Y 614.997,Z 877.154,A -85,B 0,C 180,E1 26234.155,E2 26234.155} C_VEL
LIN {X 0,Y 612.841,Z 900.81,A -85,B 0,C 180,E1 26233.422,E2 26233.422} C_VEL
LIN {X 0,Y 610.735,Z 921.176,A -85,B 0,C 180,E1 26232.67,E2 26232.67} C_VEL
LIN {X 0,Y 608.558,Z 940.534,A -85,B 0,C 180,E1 26231.84,E2 26231.84} C_VEL
LIN {X 0,Y 606.268,Z 958.983,A -85,B 0,C 180,E1 26230.943,E2 26230.943} C_VEL
LIN {X 0,Y 603.66,Z 978.532,A -85,B 0,C 180,E1 26229.866,E2 26229.866} C_VEL
LIN {X 0,Y 600.517,Z 1001.112,A -85,B 0,C 180,E1 26228.453,E2 26228.453} C_VEL
LIN {X 0,Y 597.051,Z 1024.224,A -85,B 0,C 180,E1 26226.776,E2 26226.776} C_VEL
LIN {X 0,Y 594.203,Z 1042.832,A -85,B 0,C 180,E1 26225.251,E2 26225.251} C_VEL
LIN {X 0,Y 591.55,Z 1060.162,A -85,B 0,C 180,E1 26223.669,E2 26223.669} C_VEL
LIN {X 0,Y 588.524,Z 1080.344,A -85,B 0,C 180,E1 26221.609,E2 26221.609} C_VEL
LIN {X 0,Y 585.85,Z 1098.461,A -85,B 0,C 180,E1 26219.49,E2 26219.49} C_VEL
LIN {X 0,Y 583.723,Z 1113.383,A -85,B 0,C 180,E1 26217.547,E2 26217.547} C_VEL
LIN {X 0,Y 581.679,Z 1129.285,A -85,B 0,C 180,E1 26215.232,E2 26215.232} C_VEL
LIN {X 0,Y 579.852,Z 1144.405,A -85,B 0,C 180,E1 26212.698,E2 26212.698} C_VEL
LIN {X 0,Y 578.642,Z 1155.782,A -85,B 0,C 180,E1 26210.534,E2 26210.534} C_VEL
LIN {X 0,Y 577.699,Z 1166.364,A -85,B 0,C 180,E1 26208.256,E2 26208.256} C_VEL
LIN {X 0,Y 576.865,Z 1177.39,A -85,B 0,C 180,E1 26205.479,E2 26205.479} C_VEL
LIN {X 0,Y 576.432,Z 1185.173,A -85,B 0,C 180,E1 26203.134,E2 26203.134} C_VEL
LIN {X 0,Y 576.142,Z 1191.612,A -85,B 0,C 180,E1 26200.798,E2 26200.798} C_VEL
LIN {X 0,Y 575.999,Z 1197.151,A -85,B 0,C 180,E1 26198.284,E2 26198.284} C_VEL
LIN {X 0,Y 575.933,Z 1201.427,A -85,B 0,C 180,E1 26195.579,E2 26195.579} C_VEL
LIN {X 0,Y 575.917,Z 1203.851,A -85,B 0,C 180,E1 26193.085,E2 26193.085} C_VEL
LIN {X 0,Y 575.905,Z 1204.804,A -85,B 0,C 180,E1 26190.895,E2 26190.895} C_VEL
LIN {X 0,Y 575.915,Z 1204.736,A -85,B 0,C 180,E1 26188.806,E2 26188.806} C_VEL
LIN {X 0,Y 575.913,Z 1203.509,A -85,B 0,C 180,E1 26186.417,E2 26186.417} C_VEL
LIN {X 0,Y 575.946,Z 1200.337,A -85,B 0,C 180,E1 26183.621,E2 26183.621} C_VEL
LIN {X 0,Y 576.025,Z 1195.923,A -85,B 0,C 180,E1 26181.113,E2 26181.113} C_VEL
LIN {X 0,Y 576.176,Z 1190.583,A -85,B 0,C 180,E1 26178.793,E2 26178.793} C_VEL
LIN {X 0,Y 576.569,Z 1182.685,A -85,B 0,C 180,E1 26176.052,E2 26176.052} C_VEL
LIN {X 0,Y 577.161,Z 1173.112,A -85,B 0,C 180,E1 26173.391,E2 26173.391} C_VEL
LIN {X 0,Y 577.893,Z 1164.073,A -85,B 0,C 180,E1 26171.227,E2 26171.227} C_VEL
LIN {X 0,Y 578.925,Z 1153.208,A -85,B 0,C 180,E1 26168.947,E2 26168.947} C_VEL
LIN {X 0,Y 580.564,Z 1138.275,A -85,B 0,C 180,E1 26166.234,E2 26166.234} C_VEL
LIN {X 0,Y 582.162,Z 1125.083,A -85,B 0,C 180,E1 26164.136,E2 26164.136} C_VEL
LIN {X 0,Y 584.064,Z 1111.071,A -85,B 0,C 180,E1 26162.138,E2 26162.138} C_VEL
LIN {X 0,Y 586.669,Z 1092.855,A -85,B 0,C 180,E1 26159.817,E2 26159.817} C_VEL
LIN {X 0,Y 589.384,Z 1074.495,A -85,B 0,C 180,E1 26157.776,E2 26157.776} C_VEL
LIN {X 0,Y 591.895,Z 1057.941,A -85,B 0,C 180,E1 26156.12,E2 26156.12} C_VEL
LIN {X 0,Y 594.593,Z 1040.393,A -85,B 0,C 180,E1 26154.539,E2 26154.539} C_VEL
LIN {X 0,Y 598.031,Z 1017.903,A -85,B 0,C 180,E1 26152.737,E2 26152.737} C_VEL
LIN {X 0,Y 601.141,Z 996.316,A -85,B 0,C 180,E1 26151.234,E2 26151.234} C_VEL
LIN {X 0,Y 603.894,Z 976.732,A -85,B 0,C 180,E1 26150.029,E2 26150.029} C_VEL
LIN {X 0,Y 606.433,Z 957.682,A -85,B 0,C 180,E1 26148.989,E2 26148.989} C_VEL
LIN {X 0,Y 608.832,Z 938.26,A -85,B 0,C 180,E1 26148.057,E2 26148.057} C_VEL
LIN {X 0,Y 611.335,Z 915.809,A -85,B 0,C 180,E1 26147.117,E2 26147.117} C_VEL
LIN {X 0,Y 614.033,Z 888.059,A -85,B 0,C 180,E1 26146.166,E2 26146.166} C_VEL
LIN {X 0,Y 615.868,Z 865.58,A -85,B 0,C 180,E1 26145.546,E2 26145.546} C_VEL
LIN {X 0,Y 617.295,Z 844.377,A -85,B 0,C 180,E1 26145.077,E2 26145.077} C_VEL
LIN {X 0,Y 618.445,Z 822.004,A -85,B 0,C 180,E1 26144.697,E2 26144.697} C_VEL
LIN {X 0,Y 624.381,Z 602.74,A -85,B 0,C 180,E1 26141.635,E2 26141.635} C_VEL
LIN {X 0,Y 629.775,Z 416.745,A -85,B 0,C 180,E1 26138.971,E2 26138.971} C_VEL
LIN {X 0,Y 616.934,Z 397.143,A -85,B 0,C 180,E1 26137.021,E2 26137.021} C_VEL
LIN {X 0,Y 607.519,Z 383.518,A -85,B 0,C 180,E1 26135.462,E2 26135.462} C_VEL
LIN {X 0,Y 600.22,Z 373.88,A -85,B 0,C 180,E1 26134.182,E2 26134.182} C_VEL
LIN {X 0,Y 595.824,Z 368.1,A -85,B 0,C 180,E1 26133.368,E2 26133.368} C_VEL
LIN {X 0,Y 591.756,Z 362.888,A -85,B 0,C 180,E1 26132.588,E2 26132.588} C_VEL
LIN {X 0,Y 586.161,Z 355.906,A -85,B 0,C 180,E1 26131.466,E2 26131.466} C_VEL
LIN {X 0,Y 583.278,Z 352.417,A -85,B 0,C 180,E1 26130.864,E2 26130.864} C_VEL
LIN {X 0,Y 580.362,Z 348.589,A -85,B 0,C 180,E1 26130.204,E2 26130.204} C_VEL
LIN {X 0,Y 579.763,Z 347.146,A -85,B 0,C 180,E1 26129.896,E2 26129.896} C_VEL
LIN {X 0,Y 577.664,Z 344.046,A -85,B 0,C 180,E1 26129.063,E2 26129.063} C_VEL
LIN {X 0,Y 577.266,Z 342.311,A -85,B 0,C 180,E1 26128.713,E2 26128.713} C_VEL
LIN {X 0,Y 577.26,Z 342.311,A -85,B 0,C 180,E1 26125.33,E2 26125.33} C_VEL
LIN {X 0,Y 577.286,Z 342.276,A -85,B 0,C 180,E1 26122.292,E2 26122.292} C_VEL
LIN {X 0,Y 577.259,Z 342.31,A -85,B 0,C 180,E1 26119.11,E2 26119.11} C_VEL
LIN {X 0,Y 577.306,Z 342.296,A -85,B 0,C 180,E1 26115.985,E2 26115.985} C_VEL
LIN {X 0,Y 577.251,Z 342.282,A -85,B 0,C 180,E1 26112.795,E2 26112.795} C_VEL
LIN {X 0,Y 577.319,Z 342.317,A -85,B 0,C 180,E1 26109.672,E2 26109.672} C_VEL
LIN {X 0,Y 577.252,Z 342.278,A -85,B 0,C 180,E1 26106.565,E2 26106.565} C_VEL
LIN {X 0,Y 577.319,Z 342.311,A -85,B 0,C 180,E1 26103.376,E2 26103.376} C_VEL
LIN {X 0,Y 577.254,Z 342.29,A -85,B 0,C 180,E1 26100.198,E2 26100.198} C_VEL
LIN {X 0,Y 577.308,Z 342.287,A -85,B 0,C 180,E1 26097.022,E2 26097.022} C_VEL
LIN {X 0,Y 577.261,Z 342.311,A -85,B 0,C 180,E1 26093.935,E2 26093.935} C_VEL
LIN {X 0,Y 577.298,Z 342.274,A -85,B 0,C 180,E1 26090.73,E2 26090.73} C_VEL
LIN {X 0,Y 577.272,Z 342.323,A -85,B 0,C 180,E1 26087.597,E2 26087.597} C_VEL
LIN {X 0,Y 577.271,Z 342.291,A -85,B 0,C 180,E1 26084.22,E2 26084.22} C_VEL
LIN {X 0,Y 577.285,Z 342.282,A -85,B 0,C 180,E1 26081.206,E2 26081.206} C_VEL
LIN {X 0,Y 577.269,Z 342.314,A -85,B 0,C 180,E1 26077.917,E2 26077.917} C_VEL
LIN {X 0,Y 577.271,Z 342.328,A -85,B 0,C 180,E1 26077.386,E2 26077.386} C_VEL
LIN {X 0,Y 577.722,Z 344.102,A -85,B 0,C 180,E1 26077.189,E2 26077.189} C_VEL
LIN {X 0,Y 579.588,Z 346.936,A -85,B 0,C 180,E1 26076.757,E2 26076.757} C_VEL
LIN {X 0,Y 582.504,Z 349.143,A -85,B 0,C 180,E1 26076.156,E2 26076.156} C_VEL
LIN {X 0,Y 584.723,Z 352.795,A -85,B 0,C 180,E1 26075.662,E2 26075.662} C_VEL
LIN {X 0,Y 587.82,Z 355.603,A -85,B 0,C 180,E1 26075.048,E2 26075.048} C_VEL
LIN {X 0,Y 590.728,Z 359.626,A -85,B 0,C 180,E1 26074.456,E2 26074.456} C_VEL
LIN {X 0,Y 593.21,Z 362.363,A -85,B 0,C 180,E1 26073.981,E2 26073.981} C_VEL
LIN {X 0,Y 601.347,Z 372.777,A -85,B 0,C 180,E1 26072.468,E2 26072.468} C_VEL
LIN {X 0,Y 608.276,Z 381.878,A -85,B 0,C 180,E1 26071.261,E2 26071.261} C_VEL
LIN {X 0,Y 617.428,Z 394.805,A -85,B 0,C 180,E1 26069.758,E2 26069.758} C_VEL
LIN {X 0,Y 629.736,Z 413.566,A -85,B 0,C 180,E1 26067.89,E2 26067.89} C_VEL
LIN {X 0,Y 623.765,Z 618.402,A -85,B 0,C 180,E1 26064.966,E2 26064.966} C_VEL
LIN {X 0,Y 621.23,Z 711.273,A -85,B 0,C 180,E1 26063.667,E2 26063.667} C_VEL
LIN {X 0,Y 620.318,Z 718.978,A -85,B 0,C 180,E1 26063.629,E2 26063.629} C_VEL
LIN {X 0,Y 615.469,Z 739.613,A -85,B 0,C 180,E1 26063.763,E2 26063.763} C_VEL
LIN {X 0,Y 614.777,Z 746.22,A -85,B 0,C 180,E1 26063.721,E2 26063.721} C_VEL
LIN {X 0,Y 612.545,Z 819.923,A -85,B 0,C 180,E1 26062.675,E2 26062.675} C_VEL
LIN {X 0,Y 610.783,Z 848.335,A -85,B 0,C 180,E1 26062.123,E2 26062.123} C_VEL
LIN {X 0,Y 608.774,Z 872.777,A -85,B 0,C 180,E1 26061.486,E2 26061.486} C_VEL
LIN {X 0,Y 606.325,Z 898.053,A -85,B 0,C 180,E1 26060.66,E2 26060.66} C_VEL
LIN {X 0,Y 603.301,Z 924.241,A -85,B 0,C 180,E1 26059.607,E2 26059.607} C_VEL
LIN {X 0,Y 600.412,Z 946.714,A -85,B 0,C 180,E1 26058.536,E2 26058.536} C_VEL
LIN {X 0,Y 596.85,Z 972.238,A -85,B 0,C 180,E1 26057.111,E2 26057.111} C_VEL
LIN {X 0,Y 593.715,Z 992.954,A -85,B 0,C 180,E1 26055.772,E2 26055.772} C_VEL
LIN {X 0,Y 590.814,Z 1011.534,A -85,B 0,C 180,E1 26054.423,E2 26054.423} C_VEL
LIN {X 0,Y 587.487,Z 1032.624,A -85,B 0,C 180,E1 26052.704,E2 26052.704} C_VEL
LIN {X 0,Y 583.993,Z 1053.877,A -85,B 0,C 180,E1 26050.716,E2 26050.716} C_VEL
LIN {X 0,Y 581.151,Z 1071.646,A -85,B 0,C 180,E1 26048.844,E2 26048.844} C_VEL
LIN {X 0,Y 578.135,Z 1091.286,A -85,B 0,C 180,E1 26046.508,E2 26046.508} C_VEL
LIN {X 0,Y 575.626,Z 1108.081,A -85,B 0,C 180,E1 26044.225,E2 26044.225} C_VEL
LIN {X 0,Y 573.472,Z 1124.065,A -85,B 0,C 180,E1 26041.772,E2 26041.772} C_VEL
LIN {X 0,Y 571.737,Z 1137.98,A -85,B 0,C 180,E1 26039.319,E2 26039.319} C_VEL
LIN {X 0,Y 570.383,Z 1150.611,A -85,B 0,C 180,E1 26036.776,E2 26036.776} C_VEL
LIN {X 0,Y 569.307,Z 1162.637,A -85,B 0,C 180,E1 26033.935,E2 26033.935} C_VEL
LIN {X 0,Y 568.691,Z 1171.484,A -85,B 0,C 180,E1 26031.451,E2 26031.451} C_VEL
LIN {X 0,Y 568.286,Z 1179.161,A -85,B 0,C 180,E1 26028.889,E2 26028.889} C_VEL
LIN {X 0,Y 568.046,Z 1185.57,A -85,B 0,C 180,E1 26026.147,E2 26026.147} C_VEL
LIN {X 0,Y 567.952,Z 1189.66,A -85,B 0,C 180,E1 26023.852,E2 26023.852} C_VEL
LIN {X 0,Y 567.917,Z 1192.802,A -85,B 0,C 180,E1 26021.372,E2 26021.372} C_VEL
LIN {X 0,Y 567.909,Z 1194.621,A -85,B 0,C 180,E1 26018.709,E2 26018.709} C_VEL
LIN {X 0,Y 567.912,Z 1194.856,A -85,B 0,C 180,E1 26016.267,E2 26016.267} C_VEL
LIN {X 0,Y 567.911,Z 1193.993,A -85,B 0,C 180,E1 26014.038,E2 26014.038} C_VEL
LIN {X 0,Y 567.922,Z 1191.794,A -85,B 0,C 180,E1 26011.614,E2 26011.614} C_VEL
LIN {X 0,Y 567.996,Z 1187.777,A -85,B 0,C 180,E1 26008.891,E2 26008.891} C_VEL
LIN {X 0,Y 568.13,Z 1182.485,A -85,B 0,C 180,E1 26006.368,E2 26006.368} C_VEL
LIN {X 0,Y 568.402,Z 1176.369,A -85,B 0,C 180,E1 26004.043,E2 26004.043} C_VEL
LIN {X 0,Y 568.881,Z 1168.309,A -85,B 0,C 180,E1 26001.51,E2 26001.51} C_VEL
LIN {X 0,Y 569.728,Z 1157.757,A -85,B 0,C 180,E1 25998.767,E2 25998.767} C_VEL
LIN {X 0,Y 570.761,Z 1146.754,A -85,B 0,C 180,E1 25996.32,E2 25996.32} C_VEL
LIN {X 0,Y 572.339,Z 1132.969,A -85,B 0,C 180,E1 25993.665,E2 25993.665} C_VEL
LIN {X 0,Y 574.204,Z 1118.217,A -85,B 0,C 180,E1 25991.208,E2 25991.208} C_VEL
LIN {X 0,Y 576.506,Z 1102.259,A -85,B 0,C 180,E1 25988.854,E2 25988.854} C_VEL
LIN {X 0,Y 579.078,Z 1084.822,A -85,B 0,C 180,E1 25986.601,E2 25986.601} C_VEL
LIN {X 0,Y 581.739,Z 1067.966,A -85,B 0,C 180,E1 25984.662,E2 25984.662} C_VEL
LIN {X 0,Y 585.062,Z 1047.628,A -85,B 0,C 180,E1 25982.576,E2 25982.576} C_VEL
LIN {X 0,Y 588.308,Z 1027.224,A -85,B 0,C 180,E1 25980.75,E2 25980.75} C_VEL
LIN {X 0,Y 591.334,Z 1008.205,A -85,B 0,C 180,E1 25979.232,E2 25979.232} C_VEL
LIN {X 0,Y 594.968,Z 984.805,A -85,B 0,C 180,E1 25977.582,E2 25977.582} C_VEL
LIN {X 0,Y 598.311,Z 961.755,A -85,B 0,C 180,E1 25976.187,E2 25976.187} C_VEL
LIN {X 0,Y 601.399,Z 939.269,A -85,B 0,C 180,E1 25975,E2 25975} C_VEL
LIN {X 0,Y 604.73,Z 912.211,A -85,B 0,C 180,E1 25973.793,E2 25973.793} C_VEL
LIN {X 0,Y 607.228,Z 889.083,A -85,B 0,C 180,E1 25972.94,E2 25972.94} C_VEL
LIN {X 0,Y 609.734,Z 862.236,A -85,B 0,C 180,E1 25972.127,E2 25972.127} C_VEL
LIN {X 0,Y 611.626,Z 835.651,A -85,B 0,C 180,E1 25971.517,E2 25971.517} C_VEL
LIN {X 0,Y 612.901,Z 811.647,A -85,B 0,C 180,E1 25971.107,E2 25971.107} C_VEL
LIN {X 0,Y 619.127,Z 593.967,A -85,B 0,C 180,E1 25968.044,E2 25968.044} C_VEL
LIN {X 0,Y 624.359,Z 417.549,A -85,B 0,C 180,E1 25965.514,E2 25965.514} C_VEL
LIN {X 0,Y 611.378,Z 398.877,A -85,B 0,C 180,E1 25963.676,E2 25963.676} C_VEL
LIN {X 0,Y 593.594,Z 374.712,A -85,B 0,C 180,E1 25960.971,E2 25960.971} C_VEL
LIN {X 0,Y 586.957,Z 366.247,A -85,B 0,C 180,E1 25959.895,E2 25959.895} C_VEL
LIN {X 0,Y 583.4,Z 361.549,A -85,B 0,C 180,E1 25959.293,E2 25959.293} C_VEL
LIN {X 0,Y 579.59,Z 357.154,A -85,B 0,C 180,E1 25958.647,E2 25958.647} C_VEL
LIN {X 0,Y 578.363,Z 355.403,A -85,B 0,C 180,E1 25958.427,E2 25958.427} C_VEL
LIN {X 0,Y 575.367,Z 352.35,A -85,B 0,C 180,E1 25957.909,E2 25957.909} C_VEL
LIN {X 0,Y 573.703,Z 349.464,A -85,B 0,C 180,E1 25957.59,E2 25957.59} C_VEL
LIN {X 0,Y 570.82,Z 347.083,A -85,B 0,C 180,E1 25957.086,E2 25957.086} C_VEL
LIN {X 0,Y 569.439,Z 344.143,A -85,B 0,C 180,E1 25956.8,E2 25956.8} C_VEL
LIN {X 0,Y 569.288,Z 343.311,A -85,B 0,C 180,E1 25956.738,E2 25956.738} C_VEL
LIN {X 0,Y 569.357,Z 343.309,A -85,B 0,C 180,E1 25953.587,E2 25953.587} C_VEL
LIN {X 0,Y 569.29,Z 343.318,A -85,B 0,C 180,E1 25950.387,E2 25950.387} C_VEL
LIN {X 0,Y 569.358,Z 343.253,A -85,B 0,C 180,E1 25947.282,E2 25947.282} C_VEL
LIN {X 0,Y 569.289,Z 343.314,A -85,B 0,C 180,E1 25944.157,E2 25944.157} C_VEL
LIN {X 0,Y 569.348,Z 343.252,A -85,B 0,C 180,E1 25940.994,E2 25940.994} C_VEL
LIN {X 0,Y 569.294,Z 343.316,A -85,B 0,C 180,E1 25937.901,E2 25937.901} C_VEL
LIN {X 0,Y 569.328,Z 343.31,A -85,B 0,C 180,E1 25934.61,E2 25934.61} C_VEL
